LIN {X 0,Y 360.489,Z 777.93,A -85,B 0,C 180,E1 -13047.765,E2 -13047.765} C_VEL
LIN {X 0,Y 360.532,Z 778.599,A -85,B 0,C 180,E1 -13048.883,E2 -13048.883} C_VEL
LIN {X 0,Y 360.512,Z 778.865,A -85,B 0,C 180,E1 -13050,E2 -13050} C_VEL
LIN {X 0,Y 360.53,Z 778.734,A -85,B 0,C 180,E1 -13051.117,E2 -13051.117} C_VEL
LIN {X 0,Y 360.466,Z 778.154,A -85,B 0,C 180,E1 -13052.235,E2 -13052.235} C_VEL
LIN {X 0,Y 360.409,Z 775.773,A -85,B 0,C 180,E1 -13054.474,E2 -13054.474} C_VEL
LIN {X 0,Y 360.39,Z 773.205,A -85,B 0,C 180,E1 -13055.978,E2 -13055.978} C_VEL
LIN {X 0,Y 360.621,Z 768.887,A -85,B 0,C 180,E1 -13057.841,E2 -13057.841} C_VEL
LIN {X 0,Y 360.963,Z 763.784,A -85,B 0,C 180,E1 -13059.526,E2 -13059.526} C_VEL
LIN {X 0,Y 361.5,Z 757.4,A -85,B 0,C 180,E1 -13061.21,E2 -13061.21} C_VEL
LIN {X 0,Y 362.435,Z 749.451,A -85,B 0,C 180,E1 -13062.885,E2 -13062.885} C_VEL
LIN {X 0,Y 363.324,Z 741.358,A -85,B 0,C 180,E1 -13064.278,E2 -13064.278} C_VEL
LIN {X 0,Y 364.363,Z 731.514,A -85,B 0,C 180,E1 -13065.666,E2 -13065.666} C_VEL
LIN {X 0,Y 365.512,Z 720.605,A -85,B 0,C 180,E1 -13066.907,E2 -13066.907} C_VEL
LIN {X 0,Y 366.782,Z 708.229,A -85,B 0,C 180,E1 -13067.997,E2 -13067.997} C_VEL
LIN {X 0,Y 367.813,Z 696.177,A -85,B 0,C 180,E1 -13068.81,E2 -13068.81} C_VEL
LIN {X 0,Y 368.664,Z 683.917,A -85,B 0,C 180,E1 -13069.415,E2 -13069.415} C_VEL
LIN {X 0,Y 369.374,Z 670.122,A -85,B 0,C 180,E1 -13069.846,E2 -13069.846} C_VEL
LIN {X 0,Y 370.61,Z 601.907,A -85,B 0,C 180,E1 -13071.27,E2 -13071.27} C_VEL
LIN {X 0,Y 367.336,Z 578.506,A -85,B 0,C 180,E1 -13072.019,E2 -13072.019} C_VEL
LIN {X 0,Y 364.863,Z 564.206,A -85,B 0,C 180,E1 -13072.537,E2 -13072.537} C_VEL
LIN {X 0,Y 366.628,Z 547.673,A -85,B 0,C 180,E1 -13076.16,E2 -13076.16} C_VEL
LIN {X 0,Y 365.906,Z 542.347,A -85,B 0,C 180,E1 -13077.449,E2 -13077.449} C_VEL
LIN {X 0,Y 363.599,Z 531.727,A -85,B 0,C 180,E1 -13080.168,E2 -13080.168} C_VEL
LIN {X 0,Y 361.869,Z 524.409,A -85,B 0,C 180,E1 -13082.199,E2 -13082.199} C_VEL
LIN {X 0,Y 361.868,Z 524.412,A -85,B 0,C 180,E1 -13085.636,E2 -13085.636} C_VEL
LIN {X 0,Y 361.874,Z 524.408,A -85,B 0,C 180,E1 -13089.027,E2 -13089.027} C_VEL
LIN {X 0,Y 361.882,Z 524.409,A -85,B 0,C 180,E1 -13092.439,E2 -13092.439} C_VEL
LIN {X 0,Y 361.845,Z 524.41,A -85,B 0,C 180,E1 -13095.635,E2 -13095.635} C_VEL
LIN {X 0,Y 361.833,Z 524.412,A -85,B 0,C 180,E1 -13099.243,E2 -13099.243} C_VEL
LIN {X 0,Y 361.867,Z 524.407,A -85,B 0,C 180,E1 -13102.775,E2 -13102.775} C_VEL
LIN {X 0,Y 361.85,Z 524.406,A -85,B 0,C 180,E1 -13105.719,E2 -13105.719} C_VEL
LIN {X 0,Y 361.872,Z 524.405,A -85,B 0,C 180,E1 -13109.671,E2 -13109.671} C_VEL
LIN {X 0,Y 361.949,Z 524.398,A -85,B 0,C 180,E1 -13113.474,E2 -13113.474} C_VEL
LIN {X 0,Y 361.884,Z 524.408,A -85,B 0,C 180,E1 -13117.144,E2 -13117.144} C_VEL
LIN {X 0,Y 361.9,Z 524.405,A -85,B 0,C 180,E1 -13120.722,E2 -13120.722} C_VEL
LIN {X 0,Y 361.926,Z 524.398,A -85,B 0,C 180,E1 -13123.065,E2 -13123.065} C_VEL
LIN {X 0,Y 361.992,Z 524.389,A -85,B 0,C 180,E1 -13126.527,E2 -13126.527} C_VEL
LIN {X 0,Y 362.024,Z 524.383,A -85,B 0,C 180,E1 -13129.937,E2 -13129.937} C_VEL
LIN {X 0,Y 362.16,Z 524.367,A -85,B 0,C 180,E1 -13133.313,E2 -13133.313} C_VEL
LIN {X 0,Y 362.275,Z 524.355,A -85,B 0,C 180,E1 -13137.776,E2 -13137.776} C_VEL
LIN {X 0,Y 362.421,Z 524.336,A -85,B 0,C 180,E1 -13139.999,E2 -13139.999} C_VEL
LIN {X 0,Y 362.275,Z 524.357,A -85,B 0,C 180,E1 -13142.223,E2 -13142.223} C_VEL
LIN {X 0,Y 362.16,Z 524.37,A -85,B 0,C 180,E1 -13146.686,E2 -13146.686} C_VEL
LIN {X 0,Y 362.023,Z 524.389,A -85,B 0,C 180,E1 -13150.062,E2 -13150.062} C_VEL
LIN {X 0,Y 361.989,Z 524.393,A -85,B 0,C 180,E1 -13153.898,E2 -13153.898} C_VEL
LIN {X 0,Y 361.959,Z 524.398,A -85,B 0,C 180,E1 -13157.938,E2 -13157.938} C_VEL
LIN {X 0,Y 361.883,Z 524.409,A -85,B 0,C 180,E1 -13161.653,E2 -13161.653} C_VEL
LIN {X 0,Y 361.92,Z 524.407,A -85,B 0,C 180,E1 -13165.29,E2 -13165.29} C_VEL
LIN {X 0,Y 361.916,Z 524.444,A -85,B 0,C 180,E1 -13167.856,E2 -13167.856} C_VEL
LIN {X 0,Y 362.917,Z 529.129,A -85,B 0,C 180,E1 -13169.405,E2 -13169.405} C_VEL
LIN {X 0,Y 370.573,Z 547.908,A -85,B 0,C 180,E1 -13170.406,E2 -13170.406} C_VEL
LIN {X 0,Y 371.579,Z 551.185,A -85,B 0,C 180,E1 -13170.551,E2 -13170.551} C_VEL
LIN {X 0,Y 369.705,Z 635.83,A -85,B 0,C 180,E1 -13172.34,E2 -13172.34} C_VEL
LIN {X 0,Y 369.127,Z 649.318,A -85,B 0,C 180,E1 -13172.857,E2 -13172.857} C_VEL
LIN {X 0,Y 368.497,Z 661.898,A -85,B 0,C 180,E1 -13173.578,E2 -13173.578} C_VEL
LIN {X 0,Y 367.472,Z 674.408,A -85,B 0,C 180,E1 -13174.545,E2 -13174.545} C_VEL
LIN {X 0,Y 366.504,Z 685.226,A -85,B 0,C 180,E1 -13175.623,E2 -13175.623} C_VEL
LIN {X 0,Y 365.51,Z 694.463,A -85,B 0,C 180,E1 -13176.76,E2 -13176.76} C_VEL
LIN {X 0,Y 364.419,Z 703.419,A -85,B 0,C 180,E1 -13178.106,E2 -13178.106} C_VEL
LIN {X 0,Y 363.453,Z 711.718,A -85,B 0,C 180,E1 -13179.65,E2 -13179.65} C_VEL
LIN {X 0,Y 362.559,Z 718.622,A -85,B 0,C 180,E1 -13181.228,E2 -13181.228} C_VEL
LIN {X 0,Y 361.952,Z 724.194,A -85,B 0,C 180,E1 -13182.811,E2 -13182.811} C_VEL
LIN {X 0,Y 361.396,Z 728.754,A -85,B 0,C 180,E1 -13184.433,E2 -13184.433} C_VEL
LIN {X 0,Y 360.988,Z 732.319,A -85,B 0,C 180,E1 -13186.082,E2 -13186.082} C_VEL
LIN {X 0,Y 360.669,Z 734.956,A -85,B 0,C 180,E1 -13187.77,E2 -13187.77} C_VEL
LIN {X 0,Y 360.383,Z 736.968,A -85,B 0,C 180,E1 -13189.944,E2 -13189.944} C_VEL
LIN {X 0,Y 360.299,Z 737.425,A -85,B 0,C 180,E1 -13191.378,E2 -13191.378} C_VEL
LIN {X 0,Y 360.312,Z 737.13,A -85,B 0,C 180,E1 -13193.102,E2 -13193.102} C_VEL
LIN {X 0,Y 360.444,Z 735.727,A -85,B 0,C 180,E1 -13194.976,E2 -13194.976} C_VEL
LIN {X 0,Y 360.694,Z 733.029,A -85,B 0,C 180,E1 -13196.937,E2 -13196.937} C_VEL
LIN {X 0,Y 361.096,Z 728.94,A -85,B 0,C 180,E1 -13198.91,E2 -13198.91} C_VEL
LIN {X 0,Y 361.673,Z 722.976,A -85,B 0,C 180,E1 -13200.977,E2 -13200.977} C_VEL
LIN {X 0,Y 362.343,Z 716.425,A -85,B 0,C 180,E1 -13202.729,E2 -13202.729} C_VEL
LIN {X 0,Y 362.994,Z 709.72,A -85,B 0,C 180,E1 -13204.175,E2 -13204.175} C_VEL
LIN {X 0,Y 364.002,Z 700.212,A -85,B 0,C 180,E1 -13205.828,E2 -13205.828} C_VEL
LIN {X 0,Y 364.905,Z 690.474,A -85,B 0,C 180,E1 -13207.195,E2 -13207.195} C_VEL
LIN {X 0,Y 365.774,Z 680.843,A -85,B 0,C 180,E1 -13208.293,E2 -13208.293} C_VEL
LIN {X 0,Y 366.72,Z 668.626,A -85,B 0,C 180,E1 -13209.397,E2 -13209.397} C_VEL
LIN {X 0,Y 367.467,Z 656.612,A -85,B 0,C 180,E1 -13210.228,E2 -13210.228} C_VEL
LIN {X 0,Y 368.071,Z 643.724,A -85,B 0,C 180,E1 -13210.878,E2 -13210.878} C_VEL
LIN {X 0,Y 368.446,Z 630.868,A -85,B 0,C 180,E1 -13211.296,E2 -13211.296} C_VEL
LIN {X 0,Y 369.967,Z 550.083,A -85,B 0,C 180,E1 -13212.948,E2 -13212.948} C_VEL
LIN {X 0,Y 367.904,Z 542.538,A -85,B 0,C 180,E1 -13213.224,E2 -13213.224} C_VEL
LIN {X 0,Y 362.501,Z 527.124,A -85,B 0,C 180,E1 -13213.894,E2 -13213.894} C_VEL
LIN {X 0,Y 361.982,Z 524.398,A -85,B 0,C 180,E1 -13214.733,E2 -13214.733} C_VEL
LIN {X 0,Y 361.96,Z 524.394,A -85,B 0,C 180,E1 -13217.668,E2 -13217.668} C_VEL
LIN {X 0,Y 362.142,Z 524.371,A -85,B 0,C 180,E1 -13221.782,E2 -13221.782} C_VEL
LIN {X 0,Y 362.112,Z 524.377,A -85,B 0,C 180,E1 -13224.431,E2 -13224.431} C_VEL
LIN {X 0,Y 362.28,Z 524.354,A -85,B 0,C 180,E1 -13227.776,E2 -13227.776} C_VEL
LIN {X 0,Y 362.425,Z 524.336,A -85,B 0,C 180,E1 -13230,E2 -13230} C_VEL
LIN {X 0,Y 362.28,Z 524.355,A -85,B 0,C 180,E1 -13232.224,E2 -13232.224} C_VEL
LIN {X 0,Y 362.169,Z 524.372,A -85,B 0,C 180,E1 -13236.686,E2 -13236.686} C_VEL
LIN {X 0,Y 362.071,Z 524.387,A -85,B 0,C 180,E1 -13238.933,E2 -13238.933} C_VEL
LIN {X 0,Y 361.981,Z 524.391,A -85,B 0,C 180,E1 -13240.632,E2 -13240.632} C_VEL
LIN {X 0,Y 361.285,Z 524.482,A -85,B 0,C 180,E1 -13241.561,E2 -13241.561} C_VEL
LIN {X 0,Y 358.419,Z 524.841,A -85,B 0,C 180,E1 -13243.073,E2 -13243.073} C_VEL
LIN {X 0,Y 356.005,Z 525.141,A -85,B 0,C 180,E1 -13244.295,E2 -13244.295} C_VEL
LIN {X 0,Y 354.967,Z 525.269,A -85,B 0,C 180,E1 -13245.241,E2 -13245.241} C_VEL
LIN {X 0,Y 354.881,Z 525.276,A -85,B 0,C 180,E1 -13245.562,E2 -13245.562} C_VEL
LIN {X 0,Y 354.897,Z 525.275,A -85,B 0,C 180,E1 -13248.472,E2 -13248.472} C_VEL
LIN {X 0,Y 354.83,Z 525.282,A -85,B 0,C 180,E1 -13252.106,E2 -13252.106} C_VEL
LIN {X 0,Y 354.895,Z 525.274,A -85,B 0,C 180,E1 -13255.827,E2 -13255.827} C_VEL
LIN {X 0,Y 354.849,Z 525.28,A -85,B 0,C 180,E1 -13259.678,E2 -13259.678} C_VEL
LIN {X 0,Y 354.825,Z 525.284,A -85,B 0,C 180,E1 -13263.682,E2 -13263.682} C_VEL
LIN {X 0,Y 354.796,Z 525.288,A -85,B 0,C 180,E1 -13266.459,E2 -13266.459} C_VEL
LIN {X 0,Y 354.818,Z 525.286,A -85,B 0,C 180,E1 -13269.423,E2 -13269.423} C_VEL
LIN {X 0,Y 354.835,Z 525.286,A -85,B 0,C 180,E1 -13272.876,E2 -13272.876} C_VEL
LIN {X 0,Y 354.859,Z 525.279,A -85,B 0,C 180,E1 -13276.119,E2 -13276.119} C_VEL
LIN {X 0,Y 354.849,Z 525.285,A -85,B 0,C 180,E1 -13279.188,E2 -13279.188} C_VEL
LIN {X 0,Y 354.802,Z 525.286,A -85,B 0,C 180,E1 -13282.402,E2 -13282.402} C_VEL
LIN {X 0,Y 354.805,Z 525.29,A -85,B 0,C 180,E1 -13284.941,E2 -13284.941} C_VEL
LIN {X 0,Y 354.785,Z 525.288,A -85,B 0,C 180,E1 -13288.405,E2 -13288.405} C_VEL
LIN {X 0,Y 354.846,Z 525.282,A -85,B 0,C 180,E1 -13291.619,E2 -13291.619} C_VEL
LIN {X 0,Y 354.89,Z 525.275,A -85,B 0,C 180,E1 -13294.173,E2 -13294.173} C_VEL
LIN {X 0,Y 354.808,Z 525.285,A -85,B 0,C 180,E1 -13297.893,E2 -13297.893} C_VEL
LIN {X 0,Y 354.914,Z 525.272,A -85,B 0,C 180,E1 -13301.892,E2 -13301.892} C_VEL
LIN {X 0,Y 354.935,Z 525.269,A -85,B 0,C 180,E1 -13305.981,E2 -13305.981} C_VEL
LIN {X 0,Y 354.974,Z 525.265,A -85,B 0,C 180,E1 -13309.736,E2 -13309.736} C_VEL
LIN {X 0,Y 355.106,Z 525.248,A -85,B 0,C 180,E1 -13312.037,E2 -13312.037} C_VEL
LIN {X 0,Y 355.09,Z 525.25,A -85,B 0,C 180,E1 -13314.321,E2 -13314.321} C_VEL
LIN {X 0,Y 355.238,Z 525.233,A -85,B 0,C 180,E1 -13317.733,E2 -13317.733} C_VEL
LIN {X 0,Y 355.391,Z 525.213,A -85,B 0,C 180,E1 -13320.001,E2 -13320.001} C_VEL
LIN {X 0,Y 355.246,Z 525.23,A -85,B 0,C 180,E1 -13322.268,E2 -13322.268} C_VEL
LIN {X 0,Y 355.123,Z 525.248,A -85,B 0,C 180,E1 -13326.82,E2 -13326.82} C_VEL
LIN {X 0,Y 354.971,Z 525.265,A -85,B 0,C 180,E1 -13330.265,E2 -13330.265} C_VEL
LIN {X 0,Y 354.936,Z 525.269,A -85,B 0,C 180,E1 -13334.019,E2 -13334.019} C_VEL
LIN {X 0,Y 354.916,Z 525.272,A -85,B 0,C 180,E1 -13338.109,E2 -13338.109} C_VEL
LIN {X 0,Y 354.829,Z 525.282,A -85,B 0,C 180,E1 -13342.107,E2 -13342.107} C_VEL
LIN {X 0,Y 354.894,Z 525.276,A -85,B 0,C 180,E1 -13345.828,E2 -13345.828} C_VEL
LIN {X 0,Y 354.85,Z 525.282,A -85,B 0,C 180,E1 -13349.679,E2 -13349.679} C_VEL
LIN {X 0,Y 354.827,Z 525.285,A -85,B 0,C 180,E1 -13353.683,E2 -13353.683} C_VEL
LIN {X 0,Y 354.797,Z 525.286,A -85,B 0,C 180,E1 -13356.46,E2 -13356.46} C_VEL
LIN {X 0,Y 354.821,Z 525.289,A -85,B 0,C 180,E1 -13359.425,E2 -13359.425} C_VEL
LIN {X 0,Y 354.789,Z 525.289,A -85,B 0,C 180,E1 -13362.869,E2 -13362.869} C_VEL
LIN {X 0,Y 354.839,Z 525.281,A -85,B 0,C 180,E1 -13366.116,E2 -13366.116} C_VEL
LIN {X 0,Y 354.855,Z 525.284,A -85,B 0,C 180,E1 -13369.19,E2 -13369.19} C_VEL
LIN {X 0,Y 354.809,Z 525.285,A -85,B 0,C 180,E1 -13372.403,E2 -13372.403} C_VEL
LIN {X 0,Y 354.812,Z 525.286,A -85,B 0,C 180,E1 -13374.942,E2 -13374.942} C_VEL
LIN {X 0,Y 354.825,Z 525.36,A -85,B 0,C 180,E1 -13378.398,E2 -13378.398} C_VEL
LIN {X 0,Y 357.868,Z 539.227,A -85,B 0,C 180,E1 -13381.88,E2 -13381.88} C_VEL
LIN {X 0,Y 359.195,Z 546.187,A -85,B 0,C 180,E1 -13383.559,E2 -13383.559} C_VEL
LIN {X 0,Y 358.662,Z 553.068,A -85,B 0,C 180,E1 -13385.084,E2 -13385.084} C_VEL
LIN {X 0,Y 357.409,Z 565.665,A -85,B 0,C 180,E1 -13387.836,E2 -13387.836} C_VEL
LIN {X 0,Y 362.616,Z 603.252,A -85,B 0,C 180,E1 -13388.957,E2 -13388.957} C_VEL
LIN {X 0,Y 361.342,Z 674.648,A -85,B 0,C 180,E1 -13390.471,E2 -13390.471} C_VEL
LIN {X 0,Y 360.499,Z 688.367,A -85,B 0,C 180,E1 -13390.978,E2 -13390.978} C_VEL
LIN {X 0,Y 359.661,Z 700.264,A -85,B 0,C 180,E1 -13391.634,E2 -13391.634} C_VEL
LIN {X 0,Y 358.816,Z 711.594,A -85,B 0,C 180,E1 -13392.474,E2 -13392.474} C_VEL
LIN {X 0,Y 357.599,Z 723.289,A -85,B 0,C 180,E1 -13393.59,E2 -13393.59} C_VEL
LIN {X 0,Y 356.687,Z 733.434,A -85,B 0,C 180,E1 -13394.81,E2 -13394.81} C_VEL
LIN {X 0,Y 355.685,Z 743.354,A -85,B 0,C 180,E1 -13396.284,E2 -13396.284} C_VEL
LIN {X 0,Y 354.762,Z 752.511,A -85,B 0,C 180,E1 -13397.995,E2 -13397.995} C_VEL
LIN {X 0,Y 354.099,Z 759.888,A -85,B 0,C 180,E1 -13399.71,E2 -13399.71} C_VEL
LIN {X 0,Y 353.654,Z 765.787,A -85,B 0,C 180,E1 -13401.429,E2 -13401.429} C_VEL
LIN {X 0,Y 353.431,Z 770.417,A -85,B 0,C 180,E1 -13403.148,E2 -13403.148} C_VEL
LIN {X 0,Y 353.343,Z 772.847,A -85,B 0,C 180,E1 -13404.293,E2 -13404.293} C_VEL
LIN {X 0,Y 353.351,Z 774.835,A -85,B 0,C 180,E1 -13405.437,E2 -13405.437} C_VEL
LIN {X 0,Y 353.306,Z 776.391,A -85,B 0,C 180,E1 -13406.579,E2 -13406.579} C_VEL
LIN {X 0,Y 353.39,Z 777.496,A -85,B 0,C 180,E1 -13407.721,E2 -13407.721} C_VEL
LIN {X 0,Y 353.467,Z 778.176,A -85,B 0,C 180,E1 -13408.861,E2 -13408.861} C_VEL
LIN {X 0,Y 353.448,Z 778.451,A -85,B 0,C 180,E1 -13410,E2 -13410} C_VEL
LIN {X 0,Y 353.465,Z 778.33,A -85,B 0,C 180,E1 -13411.139,E2 -13411.139} C_VEL
LIN {X 0,Y 353.367,Z 777.762,A -85,B 0,C 180,E1 -13412.28,E2 -13412.28} C_VEL
LIN {X 0,Y 353.317,Z 775.399,A -85,B 0,C 180,E1 -13414.563,E2 -13414.563} C_VEL
LIN {X 0,Y 353.316,Z 773.108,A -85,B 0,C 180,E1 -13415.965,E2 -13415.965} C_VEL
LIN {X 0,Y 353.547,Z 768.557,A -85,B 0,C 180,E1 -13417.998,E2 -13417.998} C_VEL
LIN {X 0,Y 353.94,Z 763.482,A -85,B 0,C 180,E1 -13419.717,E2 -13419.717} C_VEL
LIN {X 0,Y 354.492,Z 757.119,A -85,B 0,C 180,E1 -13421.435,E2 -13421.435} C_VEL
LIN {X 0,Y 355.49,Z 749.214,A -85,B 0,C 180,E1 -13423.141,E2 -13423.141} C_VEL
LIN {X 0,Y 356.422,Z 741.154,A -85,B 0,C 180,E1 -13424.56,E2 -13424.56} C_VEL
LIN {X 0,Y 357.521,Z 731.349,A -85,B 0,C 180,E1 -13425.974,E2 -13425.974} C_VEL
LIN {X 0,Y 358.713,Z 720.496,A -85,B 0,C 180,E1 -13427.237,E2 -13427.237} C_VEL
LIN {X 0,Y 359.886,Z 709.991,A -85,B 0,C 180,E1 -13428.207,E2 -13428.207} C_VEL
LIN {X 0,Y 360.944,Z 698.556,A -85,B 0,C 180,E1 -13429.034,E2 -13429.034} C_VEL
LIN {X 0,Y 361.885,Z 685.825,A -85,B 0,C 180,E1 -13429.72,E2 -13429.72} C_VEL
LIN {X 0,Y 362.703,Z 672.672,A -85,B 0,C 180,E1 -13430.19,E2 -13430.19} C_VEL
LIN {X 0,Y 364.152,Z 603.214,A -85,B 0,C 180,E1 -13431.678,E2 -13431.678} C_VEL
LIN {X 0,Y 360.885,Z 579.589,A -85,B 0,C 180,E1 -13432.453,E2 -13432.453} C_VEL
LIN {X 0,Y 358.112,Z 563.696,A -85,B 0,C 180,E1 -13433.061,E2 -13433.061} C_VEL
LIN {X 0,Y 359.776,Z 548.549,A -85,B 0,C 180,E1 -13436.461,E2 -13436.461} C_VEL
LIN {X 0,Y 358.156,Z 539.568,A -85,B 0,C 180,E1 -13438.733,E2 -13438.733} C_VEL
LIN {X 0,Y 355.541,Z 528.262,A -85,B 0,C 180,E1 -13441.789,E2 -13441.789} C_VEL
LIN {X 0,Y 354.814,Z 525.287,A -85,B 0,C 180,E1 -13442.666,E2 -13442.666} C_VEL
LIN {X 0,Y 354.799,Z 525.294,A -85,B 0,C 180,E1 -13446.458,E2 -13446.458} C_VEL
LIN {X 0,Y 354.823,Z 525.287,A -85,B 0,C 180,E1 -13449.423,E2 -13449.423} C_VEL
LIN {X 0,Y 354.833,Z 525.284,A -85,B 0,C 180,E1 -13452.874,E2 -13452.874} C_VEL
LIN {X 0,Y 354.782,Z 525.29,A -85,B 0,C 180,E1 -13456.105,E2 -13456.105} C_VEL
LIN {X 0,Y 354.786,Z 525.291,A -85,B 0,C 180,E1 -13459.178,E2 -13459.178} C_VEL
LIN {X 0,Y 354.809,Z 525.288,A -85,B 0,C 180,E1 -13462.4,E2 -13462.4} C_VEL
LIN {X 0,Y 354.808,Z 525.288,A -85,B 0,C 180,E1 -13464.94,E2 -13464.94} C_VEL
LIN {X 0,Y 354.789,Z 525.291,A -85,B 0,C 180,E1 -13468.404,E2 -13468.404} C_VEL
LIN {X 0,Y 354.849,Z 525.279,A -85,B 0,C 180,E1 -13471.618,E2 -13471.618} C_VEL
LIN {X 0,Y 354.894,Z 525.277,A -85,B 0,C 180,E1 -13474.172,E2 -13474.172} C_VEL
LIN {X 0,Y 354.829,Z 525.284,A -85,B 0,C 180,E1 -13477.893,E2 -13477.893} C_VEL
LIN {X 0,Y 354.916,Z 525.272,A -85,B 0,C 180,E1 -13481.891,E2 -13481.891} C_VEL
LIN {X 0,Y 354.936,Z 525.268,A -85,B 0,C 180,E1 -13485.981,E2 -13485.981} C_VEL
LIN {X 0,Y 354.971,Z 525.262,A -85,B 0,C 180,E1 -13489.735,E2 -13489.735} C_VEL
LIN {X 0,Y 355.124,Z 525.245,A -85,B 0,C 180,E1 -13493.18,E2 -13493.18} C_VEL
LIN {X 0,Y 355.238,Z 525.232,A -85,B 0,C 180,E1 -13497.732,E2 -13497.732} C_VEL
LIN {X 0,Y 355.391,Z 525.212,A -85,B 0,C 180,E1 -13499.999,E2 -13499.999} C_VEL
LIN {X 0,Y 355.239,Z 525.234,A -85,B 0,C 180,E1 -13502.267,E2 -13502.267} C_VEL
LIN {X 0,Y 355.122,Z 525.247,A -85,B 0,C 180,E1 -13506.819,E2 -13506.819} C_VEL
LIN {X 0,Y 354.97,Z 525.268,A -85,B 0,C 180,E1 -13510.264,E2 -13510.264} C_VEL
LIN {X 0,Y 354.934,Z 525.272,A -85,B 0,C 180,E1 -13514.018,E2 -13514.018} C_VEL
LIN {X 0,Y 354.914,Z 525.275,A -85,B 0,C 180,E1 -13518.108,E2 -13518.108} C_VEL
LIN {X 0,Y 354.826,Z 525.288,A -85,B 0,C 180,E1 -13522.106,E2 -13522.106} C_VEL
LIN {X 0,Y 354.891,Z 525.286,A -85,B 0,C 180,E1 -13525.827,E2 -13525.827} C_VEL
LIN {X 0,Y 354.881,Z 525.353,A -85,B 0,C 180,E1 -13527.415,E2 -13527.415} C_VEL
LIN {X 0,Y 355.808,Z 529.629,A -85,B 0,C 180,E1 -13528.861,E2 -13528.861} C_VEL
LIN {X 0,Y 364.058,Z 549.422,A -85,B 0,C 180,E1 -13529.972,E2 -13529.972} C_VEL
LIN {X 0,Y 365.108,Z 552.979,A -85,B 0,C 180,E1 -13530.13,E2 -13530.13} C_VEL
LIN {X 0,Y 363.179,Z 635.861,A -85,B 0,C 180,E1 -13531.912,E2 -13531.912} C_VEL
LIN {X 0,Y 362.54,Z 649.631,A -85,B 0,C 180,E1 -13532.445,E2 -13532.445} C_VEL
LIN {X 0,Y 361.85,Z 662.534,A -85,B 0,C 180,E1 -13533.2,E2 -13533.2} C_VEL
LIN {X 0,Y 360.885,Z 674.159,A -85,B 0,C 180,E1 -13534.112,E2 -13534.112} C_VEL
LIN {X 0,Y 359.816,Z 685.371,A -85,B 0,C 180,E1 -13535.24,E2 -13535.24} C_VEL
LIN {X 0,Y 358.654,Z 695.705,A -85,B 0,C 180,E1 -13536.544,E2 -13536.544} C_VEL
LIN {X 0,Y 357.402,Z 705.748,A -85,B 0,C 180,E1 -13538.136,E2 -13538.136} C_VEL
LIN {X 0,Y 356.366,Z 713.816,A -85,B 0,C 180,E1 -13539.726,E2 -13539.726} C_VEL
LIN {X 0,Y 355.488,Z 720.292,A -85,B 0,C 180,E1 -13541.302,E2 -13541.302} C_VEL
LIN {X 0,Y 354.864,Z 725.527,A -85,B 0,C 180,E1 -13542.882,E2 -13542.882} C_VEL
LIN {X 0,Y 354.328,Z 729.648,A -85,B 0,C 180,E1 -13544.436,E2 -13544.436} C_VEL
LIN {X 0,Y 353.934,Z 732.832,A -85,B 0,C 180,E1 -13545.975,E2 -13545.975} C_VEL
LIN {X 0,Y 353.632,Z 735.186,A -85,B 0,C 180,E1 -13547.492,E2 -13547.492} C_VEL
LIN {X 0,Y 353.387,Z 736.867,A -85,B 0,C 180,E1 -13549.088,E2 -13549.088} C_VEL
LIN {X 0,Y 353.225,Z 737.791,A -85,B 0,C 180,E1 -13550.892,E2 -13550.892} C_VEL
LIN {X 0,Y 353.222,Z 737.698,A -85,B 0,C 180,E1 -13552.737,E2 -13552.737} C_VEL
LIN {X 0,Y 353.33,Z 736.363,A -85,B 0,C 180,E1 -13554.773,E2 -13554.773} C_VEL
LIN {X 0,Y 353.527,Z 734.055,A -85,B 0,C 180,E1 -13556.609,E2 -13556.609} C_VEL
LIN {X 0,Y 353.967,Z 730.222,A -85,B 0,C 180,E1 -13558.622,E2 -13558.622} C_VEL
LIN {X 0,Y 354.345,Z 725.964,A -85,B 0,C 180,E1 -13560.275,E2 -13560.275} C_VEL
LIN {X 0,Y 355.07,Z 719.266,A -85,B 0,C 180,E1 -13562.282,E2 -13562.282} C_VEL
LIN {X 0,Y 355.832,Z 712.229,A -85,B 0,C 180,E1 -13563.931,E2 -13563.931} C_VEL
LIN {X 0,Y 356.746,Z 703.616,A -85,B 0,C 180,E1 -13565.563,E2 -13565.563} C_VEL
LIN {X 0,Y 357.725,Z 694.207,A -85,B 0,C 180,E1 -13567.006,E2 -13567.006} C_VEL
LIN {X 0,Y 358.662,Z 683.745,A -85,B 0,C 180,E1 -13568.294,E2 -13568.294} C_VEL
LIN {X 0,Y 359.646,Z 672.39,A -85,B 0,C 180,E1 -13569.406,E2 -13569.406} C_VEL
LIN {X 0,Y 360.479,Z 659.888,A -85,B 0,C 180,E1 -13570.356,E2 -13570.356} C_VEL
LIN {X 0,Y 361.132,Z 646.613,A -85,B 0,C 180,E1 -13571.087,E2 -13571.087} C_VEL
LIN {X 0,Y 361.607,Z 633.983,A -85,B 0,C 180,E1 -13571.553,E2 -13571.553} C_VEL
LIN {X 0,Y 363.192,Z 550.766,A -85,B 0,C 180,E1 -13573.308,E2 -13573.308} C_VEL
LIN {X 0,Y 359.766,Z 539.781,A -85,B 0,C 180,E1 -13573.747,E2 -13573.747} C_VEL
LIN {X 0,Y 355.361,Z 527.561,A -85,B 0,C 180,E1 -13574.295,E2 -13574.295} C_VEL
LIN {X 0,Y 354.915,Z 525.276,A -85,B 0,C 180,E1 -13575.01,E2 -13575.01} C_VEL
LIN {X 0,Y 354.932,Z 525.273,A -85,B 0,C 180,E1 -13578.58,E2 -13578.58} C_VEL
LIN {X 0,Y 355.081,Z 525.251,A -85,B 0,C 180,E1 -13582.036,E2 -13582.036} C_VEL
LIN {X 0,Y 355.086,Z 525.251,A -85,B 0,C 180,E1 -13584.321,E2 -13584.321} C_VEL
LIN {X 0,Y 355.243,Z 525.231,A -85,B 0,C 180,E1 -13587.732,E2 -13587.732} C_VEL
LIN {X 0,Y 355.395,Z 525.212,A -85,B 0,C 180,E1 -13590,E2 -13590} C_VEL
LIN {X 0,Y 355.243,Z 525.231,A -85,B 0,C 180,E1 -13592.268,E2 -13592.268} C_VEL
LIN {X 0,Y 355.135,Z 525.249,A -85,B 0,C 180,E1 -13596.819,E2 -13596.819} C_VEL
LIN {X 0,Y 355.012,Z 525.264,A -85,B 0,C 180,E1 -13599.112,E2 -13599.112} C_VEL
LIN {X 0,Y 354.918,Z 525.274,A -85,B 0,C 180,E1 -13602.581,E2 -13602.581} C_VEL
LIN {X 0,Y 354.881,Z 525.276,A -85,B 0,C 180,E1 -13605.562,E2 -13605.562} C_VEL
LIN {X 0,Y 354.204,Z 525.364,A -85,B 0,C 180,E1 -13606.51,E2 -13606.51} C_VEL
LIN {X 0,Y 351.337,Z 525.717,A -85,B 0,C 180,E1 -13608.052,E2 -13608.052} C_VEL
LIN {X 0,Y 348.913,Z 526.022,A -85,B 0,C 180,E1 -13609.299,E2 -13609.299} C_VEL
LIN {X 0,Y 347.875,Z 526.149,A -85,B 0,C 180,E1 -13610.265,E2 -13610.265} C_VEL
LIN {X 0,Y 347.792,Z 526.158,A -85,B 0,C 180,E1 -13610.592,E2 -13610.592} C_VEL
LIN {X 0,Y 347.812,Z 526.159,A -85,B 0,C 180,E1 -13614.595,E2 -13614.595} C_VEL
LIN {X 0,Y 347.808,Z 526.158,A -85,B 0,C 180,E1 -13617.693,E2 -13617.693} C_VEL
LIN {X 0,Y 347.766,Z 526.163,A -85,B 0,C 180,E1 -13620.345,E2 -13620.345} C_VEL
LIN {X 0,Y 347.743,Z 526.165,A -85,B 0,C 180,E1 -13624.044,E2 -13624.044} C_VEL
LIN {X 0,Y 347.761,Z 526.166,A -85,B 0,C 180,E1 -13627.32,E2 -13627.32} C_VEL
LIN {X 0,Y 347.787,Z 526.16,A -85,B 0,C 180,E1 -13630.288,E2 -13630.288} C_VEL
LIN {X 0,Y 347.812,Z 526.159,A -85,B 0,C 180,E1 -13633.393,E2 -13633.393} C_VEL
LIN {X 0,Y 347.81,Z 526.159,A -85,B 0,C 180,E1 -13636.67,E2 -13636.67} C_VEL
LIN {X 0,Y 347.778,Z 526.161,A -85,B 0,C 180,E1 -13640.165,E2 -13640.165} C_VEL
LIN {X 0,Y 347.781,Z 526.16,A -85,B 0,C 180,E1 -13644.125,E2 -13644.125} C_VEL
LIN {X 0,Y 347.731,Z 526.167,A -85,B 0,C 180,E1 -13648.086,E2 -13648.086} C_VEL
LIN {X 0,Y 347.799,Z 526.163,A -85,B 0,C 180,E1 -13650.99,E2 -13650.99} C_VEL
LIN {X 0,Y 347.823,Z 526.157,A -85,B 0,C 180,E1 -13653.608,E2 -13653.608} C_VEL
LIN {X 0,Y 347.777,Z 526.161,A -85,B 0,C 180,E1 -13656.162,E2 -13656.162} C_VEL
LIN {X 0,Y 347.798,Z 526.159,A -85,B 0,C 180,E1 -13659.909,E2 -13659.909} C_VEL
LIN {X 0,Y 347.858,Z 526.151,A -85,B 0,C 180,E1 -13662.359,E2 -13662.359} C_VEL
LIN {X 0,Y 347.889,Z 526.147,A -85,B 0,C 180,E1 -13665.971,E2 -13665.971} C_VEL
LIN {X 0,Y 347.925,Z 526.145,A -85,B 0,C 180,E1 -13669.526,E2 -13669.526} C_VEL
LIN {X 0,Y 348.066,Z 526.125,A -85,B 0,C 180,E1 -13671.875,E2 -13671.875} C_VEL
LIN {X 0,Y 348.065,Z 526.125,A -85,B 0,C 180,E1 -13674.206,E2 -13674.206} C_VEL
LIN {X 0,Y 348.201,Z 526.11,A -85,B 0,C 180,E1 -13677.687,E2 -13677.687} C_VEL
LIN {X 0,Y 348.361,Z 526.088,A -85,B 0,C 180,E1 -13680.001,E2 -13680.001} C_VEL
LIN {X 0,Y 348.209,Z 526.107,A -85,B 0,C 180,E1 -13682.314,E2 -13682.314} C_VEL
LIN {X 0,Y 348.088,Z 526.126,A -85,B 0,C 180,E1 -13686.959,E2 -13686.959} C_VEL
LIN {X 0,Y 347.922,Z 526.143,A -85,B 0,C 180,E1 -13690.475,E2 -13690.475} C_VEL
LIN {X 0,Y 347.892,Z 526.146,A -85,B 0,C 180,E1 -13694.151,E2 -13694.151} C_VEL
LIN {X 0,Y 347.884,Z 526.147,A -85,B 0,C 180,E1 -13698.291,E2 -13698.291} C_VEL
LIN {X 0,Y 347.783,Z 526.163,A -85,B 0,C 180,E1 -13701.636,E2 -13701.636} C_VEL
LIN {X 0,Y 347.807,Z 526.161,A -85,B 0,C 180,E1 -13705.109,E2 -13705.109} C_VEL
LIN {X 0,Y 347.807,Z 526.159,A -85,B 0,C 180,E1 -13707.695,E2 -13707.695} C_VEL
LIN {X 0,Y 347.766,Z 526.162,A -85,B 0,C 180,E1 -13710.347,E2 -13710.347} C_VEL
LIN {X 0,Y 347.744,Z 526.165,A -85,B 0,C 180,E1 -13714.045,E2 -13714.045} C_VEL
LIN {X 0,Y 347.762,Z 526.169,A -85,B 0,C 180,E1 -13717.321,E2 -13717.321} C_VEL
LIN {X 0,Y 347.73,Z 526.167,A -85,B 0,C 180,E1 -13720.298,E2 -13720.298} C_VEL
LIN {X 0,Y 347.727,Z 526.173,A -85,B 0,C 180,E1 -13723.408,E2 -13723.408} C_VEL
LIN {X 0,Y 347.781,Z 526.161,A -85,B 0,C 180,E1 -13726.677,E2 -13726.677} C_VEL
LIN {X 0,Y 347.785,Z 526.16,A -85,B 0,C 180,E1 -13730.166,E2 -13730.166} C_VEL
LIN {X 0,Y 347.789,Z 526.16,A -85,B 0,C 180,E1 -13734.126,E2 -13734.126} C_VEL
LIN {X 0,Y 347.784,Z 526.305,A -85,B 0,C 180,E1 -13738.075,E2 -13738.075} C_VEL
LIN {X 0,Y 350.807,Z 540.039,A -85,B 0,C 180,E1 -13741.604,E2 -13741.604} C_VEL
LIN {X 0,Y 352.273,Z 548.524,A -85,B 0,C 180,E1 -13743.68,E2 -13743.68} C_VEL
LIN {X 0,Y 350.822,Z 562.85,A -85,B 0,C 180,E1 -13746.888,E2 -13746.888} C_VEL
LIN {X 0,Y 350.562,Z 565.347,A -85,B 0,C 180,E1 -13747.432,E2 -13747.432} C_VEL
LIN {X 0,Y 355.879,Z 604.297,A -85,B 0,C 180,E1 -13748.621,E2 -13748.621} C_VEL
LIN {X 0,Y 354.529,Z 674.942,A -85,B 0,C 180,E1 -13750.156,E2 -13750.156} C_VEL
LIN {X 0,Y 353.676,Z 688.432,A -85,B 0,C 180,E1 -13750.672,E2 -13750.672} C_VEL
LIN {X 0,Y 352.828,Z 700.21,A -85,B 0,C 180,E1 -13751.341,E2 -13751.341} C_VEL
LIN {X 0,Y 351.864,Z 712.234,A -85,B 0,C 180,E1 -13752.266,E2 -13752.266} C_VEL
LIN {X 0,Y 350.61,Z 723.739,A -85,B 0,C 180,E1 -13753.403,E2 -13753.403} C_VEL
LIN {X 0,Y 349.693,Z 733.488,A -85,B 0,C 180,E1 -13754.613,E2 -13754.613} C_VEL
LIN {X 0,Y 348.765,Z 742.666,A -85,B 0,C 180,E1 -13756.007,E2 -13756.007} C_VEL
LIN {X 0,Y 347.756,Z 751.879,A -85,B 0,C 180,E1 -13757.749,E2 -13757.749} C_VEL
LIN {X 0,Y 347.042,Z 759.3,A -85,B 0,C 180,E1 -13759.499,E2 -13759.499} C_VEL
LIN {X 0,Y 346.61,Z 765.244,A -85,B 0,C 180,E1 -13761.253,E2 -13761.253} C_VEL
LIN {X 0,Y 346.374,Z 769.91,A -85,B 0,C 180,E1 -13763.008,E2 -13763.008} C_VEL
LIN {X 0,Y 346.233,Z 773.438,A -85,B 0,C 180,E1 -13764.759,E2 -13764.759} C_VEL
LIN {X 0,Y 346.226,Z 775.931,A -85,B 0,C 180,E1 -13766.509,E2 -13766.509} C_VEL
LIN {X 0,Y 346.293,Z 777.058,A -85,B 0,C 180,E1 -13767.674,E2 -13767.674} C_VEL
LIN {X 0,Y 346.385,Z 777.749,A -85,B 0,C 180,E1 -13768.837,E2 -13768.837} C_VEL
LIN {X 0,Y 346.385,Z 778.036,A -85,B 0,C 180,E1 -13770,E2 -13770} C_VEL
LIN {X 0,Y 346.382,Z 777.924,A -85,B 0,C 180,E1 -13771.163,E2 -13771.163} C_VEL
LIN {X 0,Y 346.268,Z 777.377,A -85,B 0,C 180,E1 -13772.326,E2 -13772.326} C_VEL
LIN {X 0,Y 346.229,Z 775.033,A -85,B 0,C 180,E1 -13774.657,E2 -13774.657} C_VEL
LIN {X 0,Y 346.283,Z 772.153,A -85,B 0,C 180,E1 -13776.408,E2 -13776.408} C_VEL
LIN {X 0,Y 346.496,Z 768.232,A -85,B 0,C 180,E1 -13778.162,E2 -13778.162} C_VEL
LIN {X 0,Y 346.902,Z 763.177,A -85,B 0,C 180,E1 -13779.916,E2 -13779.916} C_VEL
LIN {X 0,Y 347.502,Z 756.839,A -85,B 0,C 180,E1 -13781.668,E2 -13781.668} C_VEL
LIN {X 0,Y 348.546,Z 748.977,A -85,B 0,C 180,E1 -13783.408,E2 -13783.408} C_VEL
LIN {X 0,Y 349.696,Z 739.148,A -85,B 0,C 180,E1 -13785.145,E2 -13785.145} C_VEL
LIN {X 0,Y 350.924,Z 729.051,A -85,B 0,C 180,E1 -13786.582,E2 -13786.582} C_VEL
LIN {X 0,Y 352.27,Z 717.674,A -85,B 0,C 180,E1 -13787.862,E2 -13787.862} C_VEL
LIN {X 0,Y 353.452,Z 706.582,A -85,B 0,C 180,E1 -13788.851,E2 -13788.851} C_VEL
LIN {X 0,Y 354.595,Z 694.349,A -85,B 0,C 180,E1 -13789.69,E2 -13789.69} C_VEL
LIN {X 0,Y 355.588,Z 681.588,A -85,B 0,C 180,E1 -13790.31,E2 -13790.31} C_VEL
LIN {X 0,Y 356.272,Z 668.433,A -85,B 0,C 180,E1 -13790.722,E2 -13790.722} C_VEL
LIN {X 0,Y 357.575,Z 603.339,A -85,B 0,C 180,E1 -13792.14,E2 -13792.14} C_VEL
LIN {X 0,Y 354.137,Z 578.578,A -85,B 0,C 180,E1 -13792.98,E2 -13792.98} C_VEL
LIN {X 0,Y 351.35,Z 563.309,A -85,B 0,C 180,E1 -13793.581,E2 -13793.581} C_VEL
LIN {X 0,Y 352.879,Z 549.82,A -85,B 0,C 180,E1 -13796.682,E2 -13796.682} C_VEL
LIN {X 0,Y 350.929,Z 539.488,A -85,B 0,C 180,E1 -13799.383,E2 -13799.383} C_VEL
LIN {X 0,Y 348.062,Z 527.452,A -85,B 0,C 180,E1 -13802.766,E2 -13802.766} C_VEL
LIN {X 0,Y 347.783,Z 526.166,A -85,B 0,C 180,E1 -13803.147,E2 -13803.147} C_VEL
LIN {X 0,Y 347.771,Z 526.168,A -85,B 0,C 180,E1 -13806.064,E2 -13806.064} C_VEL
LIN {X 0,Y 347.785,Z 526.164,A -85,B 0,C 180,E1 -13809.834,E2 -13809.834} C_VEL
LIN {X 0,Y 347.784,Z 526.163,A -85,B 0,C 180,E1 -13813.397,E2 -13813.397} C_VEL
LIN {X 0,Y 347.728,Z 526.172,A -85,B 0,C 180,E1 -13816.684,E2 -13816.684} C_VEL
LIN {X 0,Y 347.744,Z 526.165,A -85,B 0,C 180,E1 -13820.172,E2 -13820.172} C_VEL
LIN {X 0,Y 347.762,Z 526.164,A -85,B 0,C 180,E1 -13822.679,E2 -13822.679} C_VEL
LIN {X 0,Y 347.744,Z 526.163,A -85,B 0,C 180,E1 -13825.955,E2 -13825.955} C_VEL
LIN {X 0,Y 347.76,Z 526.163,A -85,B 0,C 180,E1 -13829.653,E2 -13829.653} C_VEL
LIN {X 0,Y 347.848,Z 526.152,A -85,B 0,C 180,E1 -13832.743,E2 -13832.743} C_VEL
LIN {X 0,Y 347.783,Z 526.156,A -85,B 0,C 180,E1 -13836.161,E2 -13836.161} C_VEL
LIN {X 0,Y 347.806,Z 526.156,A -85,B 0,C 180,E1 -13839.908,E2 -13839.908} C_VEL
LIN {X 0,Y 347.86,Z 526.151,A -85,B 0,C 180,E1 -13842.358,E2 -13842.358} C_VEL
LIN {X 0,Y 347.891,Z 526.146,A -85,B 0,C 180,E1 -13845.97,E2 -13845.97} C_VEL
LIN {X 0,Y 347.922,Z 526.141,A -85,B 0,C 180,E1 -13849.525,E2 -13849.525} C_VEL
LIN {X 0,Y 348.089,Z 526.122,A -85,B 0,C 180,E1 -13853.041,E2 -13853.041} C_VEL
LIN {X 0,Y 348.201,Z 526.109,A -85,B 0,C 180,E1 -13857.686,E2 -13857.686} C_VEL
LIN {X 0,Y 348.361,Z 526.087,A -85,B 0,C 180,E1 -13859.999,E2 -13859.999} C_VEL
LIN {X 0,Y 348.201,Z 526.111,A -85,B 0,C 180,E1 -13862.313,E2 -13862.313} C_VEL
LIN {X 0,Y 348.087,Z 526.124,A -85,B 0,C 180,E1 -13866.957,E2 -13866.957} C_VEL
LIN {X 0,Y 347.92,Z 526.147,A -85,B 0,C 180,E1 -13870.474,E2 -13870.474} C_VEL
LIN {X 0,Y 347.89,Z 526.149,A -85,B 0,C 180,E1 -13874.15,E2 -13874.15} C_VEL
LIN {X 0,Y 347.882,Z 526.151,A -85,B 0,C 180,E1 -13878.29,E2 -13878.29} C_VEL
LIN {X 0,Y 347.78,Z 526.166,A -85,B 0,C 180,E1 -13881.635,E2 -13881.635} C_VEL
LIN {X 0,Y 347.804,Z 526.164,A -85,B 0,C 180,E1 -13885.108,E2 -13885.108} C_VEL
LIN {X 0,Y 347.837,Z 526.259,A -85,B 0,C 180,E1 -13886.94,E2 -13886.94} C_VEL
LIN {X 0,Y 348.771,Z 530.36,A -85,B 0,C 180,E1 -13888.305,E2 -13888.305} C_VEL
LIN {X 0,Y 357.168,Z 550.02,A -85,B 0,C 180,E1 -13889.467,E2 -13889.467} C_VEL
LIN {X 0,Y 358.543,Z 553.771,A -85,B 0,C 180,E1 -13889.663,E2 -13889.663} C_VEL
LIN {X 0,Y 356.634,Z 636.32,A -85,B 0,C 180,E1 -13891.481,E2 -13891.481} C_VEL
LIN {X 0,Y 355.964,Z 650.15,A -85,B 0,C 180,E1 -13892.026,E2 -13892.026} C_VEL
LIN {X 0,Y 355.265,Z 662.916,A -85,B 0,C 180,E1 -13892.788,E2 -13892.788} C_VEL
LIN {X 0,Y 354.217,Z 674.908,A -85,B 0,C 180,E1 -13893.748,E2 -13893.748} C_VEL
LIN {X 0,Y 353.113,Z 685.911,A -85,B 0,C 180,E1 -13894.878,E2 -13894.878} C_VEL
LIN {X 0,Y 351.976,Z 695.412,A -85,B 0,C 180,E1 -13896.088,E2 -13896.088} C_VEL
LIN {X 0,Y 350.642,Z 705.411,A -85,B 0,C 180,E1 -13897.677,E2 -13897.677} C_VEL
LIN {X 0,Y 349.577,Z 713.538,A -85,B 0,C 180,E1 -13899.286,E2 -13899.286} C_VEL
LIN {X 0,Y 348.623,Z 720.166,A -85,B 0,C 180,E1 -13900.9,E2 -13900.9} C_VEL
LIN {X 0,Y 347.784,Z 726.675,A -85,B 0,C 180,E1 -13902.918,E2 -13902.918} C_VEL
LIN {X 0,Y 347.104,Z 731.967,A -85,B 0,C 180,E1 -13905.125,E2 -13905.125} C_VEL
LIN {X 0,Y 346.67,Z 734.948,A -85,B 0,C 180,E1 -13906.871,E2 -13906.871} C_VEL
LIN {X 0,Y 346.358,Z 736.993,A -85,B 0,C 180,E1 -13908.656,E2 -13908.656} C_VEL
LIN {X 0,Y 346.132,Z 738.225,A -85,B 0,C 180,E1 -13910.993,E2 -13910.993} C_VEL
LIN {X 0,Y 346.123,Z 738.167,A -85,B 0,C 180,E1 -13912.473,E2 -13912.473} C_VEL
LIN {X 0,Y 346.199,Z 737.206,A -85,B 0,C 180,E1 -13914.292,E2 -13914.292} C_VEL
LIN {X 0,Y 346.39,Z 735.024,A -85,B 0,C 180,E1 -13916.289,E2 -13916.289} C_VEL
LIN {X 0,Y 346.814,Z 731.451,A -85,B 0,C 180,E1 -13918.331,E2 -13918.331} C_VEL
LIN {X 0,Y 347.337,Z 726.176,A -85,B 0,C 180,E1 -13920.464,E2 -13920.464} C_VEL
LIN {X 0,Y 348.001,Z 720.119,A -85,B 0,C 180,E1 -13922.323,E2 -13922.323} C_VEL
LIN {X 0,Y 348.791,Z 713.176,A -85,B 0,C 180,E1 -13924.008,E2 -13924.008} C_VEL
LIN {X 0,Y 349.712,Z 704.675,A -85,B 0,C 180,E1 -13925.671,E2 -13925.671} C_VEL
LIN {X 0,Y 350.747,Z 695.169,A -85,B 0,C 180,E1 -13927.176,E2 -13927.176} C_VEL
LIN {X 0,Y 351.684,Z 685.162,A -85,B 0,C 180,E1 -13928.457,E2 -13928.457} C_VEL
LIN {X 0,Y 352.744,Z 673.711,A -85,B 0,C 180,E1 -13929.619,E2 -13929.619} C_VEL
LIN {X 0,Y 353.573,Z 661.992,A -85,B 0,C 180,E1 -13930.553,E2 -13930.553} C_VEL
LIN {X 0,Y 354.292,Z 649.216,A -85,B 0,C 180,E1 -13931.308,E2 -13931.308} C_VEL
LIN {X 0,Y 354.821,Z 635.674,A -85,B 0,C 180,E1 -13931.848,E2 -13931.848} C_VEL
LIN {X 0,Y 355.84,Z 588.088,A -85,B 0,C 180,E1 -13932.888,E2 -13932.888} C_VEL
LIN {X 0,Y 356.527,Z 551.911,A -85,B 0,C 180,E1 -13933.661,E2 -13933.661} C_VEL
LIN {X 0,Y 350.987,Z 535.554,A -85,B 0,C 180,E1 -13934.363,E2 -13934.363} C_VEL
LIN {X 0,Y 348.23,Z 527.955,A -85,B 0,C 180,E1 -13934.722,E2 -13934.722} C_VEL
LIN {X 0,Y 347.909,Z 526.146,A -85,B 0,C 180,E1 -13935.3,E2 -13935.3} C_VEL
LIN {X 0,Y 347.882,Z 526.149,A -85,B 0,C 180,E1 -13938.345,E2 -13938.345} C_VEL
LIN {X 0,Y 348.043,Z 526.128,A -85,B 0,C 180,E1 -13941.874,E2 -13941.874} C_VEL
LIN {X 0,Y 348.06,Z 526.126,A -85,B 0,C 180,E1 -13944.206,E2 -13944.206} C_VEL
LIN {X 0,Y 348.206,Z 526.108,A -85,B 0,C 180,E1 -13947.687,E2 -13947.687} C_VEL
LIN {X 0,Y 348.344,Z 526.09,A -85,B 0,C 180,E1 -13950,E2 -13950} C_VEL
LIN {X 0,Y 348.205,Z 526.108,A -85,B 0,C 180,E1 -13952.313,E2 -13952.313} C_VEL
LIN {X 0,Y 348.104,Z 526.126,A -85,B 0,C 180,E1 -13956.958,E2 -13956.958} C_VEL
LIN {X 0,Y 347.964,Z 526.14,A -85,B 0,C 180,E1 -13959.298,E2 -13959.298} C_VEL
LIN {X 0,Y 347.886,Z 526.152,A -85,B 0,C 180,E1 -13962.839,E2 -13962.839} C_VEL
LIN {X 0,Y 347.835,Z 526.155,A -85,B 0,C 180,E1 -13966.431,E2 -13966.431} C_VEL
LIN {X 0,Y 347.847,Z 526.157,A -85,B 0,C 180,E1 -13968.86,E2 -13968.86} C_VEL
LIN {X 0,Y 347.792,Z 526.158,A -85,B 0,C 180,E1 -13970.592,E2 -13970.592} C_VEL
LIN {X 0,Y 347.136,Z 526.243,A -85,B 0,C 180,E1 -13971.558,E2 -13971.558} C_VEL
LIN {X 0,Y 344.31,Z 526.598,A -85,B 0,C 180,E1 -13973.129,E2 -13973.129} C_VEL
LIN {X 0,Y 341.904,Z 526.897,A -85,B 0,C 180,E1 -13974.401,E2 -13974.401} C_VEL
LIN {X 0,Y 340.858,Z 527.026,A -85,B 0,C 180,E1 -13975.385,E2 -13975.385} C_VEL
LIN {X 0,Y 340.766,Z 527.035,A -85,B 0,C 180,E1 -13975.718,E2 -13975.718} C_VEL
LIN {X 0,Y 340.738,Z 527.038,A -85,B 0,C 180,E1 -13978.319,E2 -13978.319} C_VEL
LIN {X 0,Y 340.711,Z 527.047,A -85,B 0,C 180,E1 -13981.042,E2 -13981.042} C_VEL
LIN {X 0,Y 340.713,Z 527.044,A -85,B 0,C 180,E1 -13985.278,E2 -13985.278} C_VEL
LIN {X 0,Y 340.714,Z 527.041,A -85,B 0,C 180,E1 -13988.388,E2 -13988.388} C_VEL
LIN {X 0,Y 340.72,Z 527.044,A -85,B 0,C 180,E1 -13991.303,E2 -13991.303} C_VEL
LIN {X 0,Y 340.774,Z 527.034,A -85,B 0,C 180,E1 -13994.522,E2 -13994.522} C_VEL
LIN {X 0,Y 340.745,Z 527.037,A -85,B 0,C 180,E1 -13997.945,E2 -13997.945} C_VEL
LIN {X 0,Y 340.727,Z 527.039,A -85,B 0,C 180,E1 -14000.252,E2 -14000.252} C_VEL
LIN {X 0,Y 340.703,Z 527.044,A -85,B 0,C 180,E1 -14003.559,E2 -14003.559} C_VEL
LIN {X 0,Y 340.685,Z 527.044,A -85,B 0,C 180,E1 -14006.153,E2 -14006.153} C_VEL
LIN {X 0,Y 340.767,Z 527.034,A -85,B 0,C 180,E1 -14010.332,E2 -14010.332} C_VEL
LIN {X 0,Y 340.797,Z 527.036,A -85,B 0,C 180,E1 -14013.02,E2 -14013.02} C_VEL
LIN {X 0,Y 340.746,Z 527.038,A -85,B 0,C 180,E1 -14015.638,E2 -14015.638} C_VEL
LIN {X 0,Y 340.726,Z 527.042,A -85,B 0,C 180,E1 -14019.474,E2 -14019.474} C_VEL
LIN {X 0,Y 340.849,Z 527.024,A -85,B 0,C 180,E1 -14021.984,E2 -14021.984} C_VEL
LIN {X 0,Y 340.861,Z 527.024,A -85,B 0,C 180,E1 -14025.705,E2 -14025.705} C_VEL
LIN {X 0,Y 340.867,Z 527.026,A -85,B 0,C 180,E1 -14029.307,E2 -14029.307} C_VEL
LIN {X 0,Y 341.07,Z 527,A -85,B 0,C 180,E1 -14032.899,E2 -14032.899} C_VEL
LIN {X 0,Y 341.163,Z 526.987,A -85,B 0,C 180,E1 -14037.639,E2 -14037.639} C_VEL
LIN {X 0,Y 341.309,Z 526.967,A -85,B 0,C 180,E1 -14040.001,E2 -14040.001} C_VEL
LIN {X 0,Y 341.171,Z 526.984,A -85,B 0,C 180,E1 -14042.362,E2 -14042.362} C_VEL
LIN {X 0,Y 341.055,Z 527.003,A -85,B 0,C 180,E1 -14047.103,E2 -14047.103} C_VEL
LIN {X 0,Y 340.864,Z 527.023,A -85,B 0,C 180,E1 -14050.695,E2 -14050.695} C_VEL
LIN {X 0,Y 340.857,Z 527.023,A -85,B 0,C 180,E1 -14054.326,E2 -14054.326} C_VEL
LIN {X 0,Y 340.831,Z 527.026,A -85,B 0,C 180,E1 -14058.467,E2 -14058.467} C_VEL
LIN {X 0,Y 340.748,Z 527.037,A -85,B 0,C 180,E1 -14061.858,E2 -14061.858} C_VEL
LIN {X 0,Y 340.768,Z 527.036,A -85,B 0,C 180,E1 -14065.665,E2 -14065.665} C_VEL
LIN {X 0,Y 340.738,Z 527.038,A -85,B 0,C 180,E1 -14068.321,E2 -14068.321} C_VEL
LIN {X 0,Y 340.712,Z 527.044,A -85,B 0,C 180,E1 -14071.044,E2 -14071.044} C_VEL
LIN {X 0,Y 340.715,Z 527.047,A -85,B 0,C 180,E1 -14075.28,E2 -14075.28} C_VEL
LIN {X 0,Y 340.709,Z 527.041,A -85,B 0,C 180,E1 -14078.388,E2 -14078.388} C_VEL
LIN {X 0,Y 340.697,Z 527.043,A -85,B 0,C 180,E1 -14082.047,E2 -14082.047} C_VEL
LIN {X 0,Y 340.719,Z 527.045,A -85,B 0,C 180,E1 -14085.469,E2 -14085.469} C_VEL
LIN {X 0,Y 340.724,Z 527.04,A -85,B 0,C 180,E1 -14088.697,E2 -14088.697} C_VEL
LIN {X 0,Y 340.739,Z 527.04,A -85,B 0,C 180,E1 -14091.775,E2 -14091.775} C_VEL
LIN {X 0,Y 340.723,Z 527.045,A -85,B 0,C 180,E1 -14095.596,E2 -14095.596} C_VEL
LIN {X 0,Y 340.746,Z 527.239,A -85,B 0,C 180,E1 -14097.741,E2 -14097.741} C_VEL
LIN {X 0,Y 343.561,Z 540.107,A -85,B 0,C 180,E1 -14101.125,E2 -14101.125} C_VEL
LIN {X 0,Y 345.29,Z 549.127,A -85,B 0,C 180,E1 -14103.399,E2 -14103.399} C_VEL
LIN {X 0,Y 344.204,Z 560.031,A -85,B 0,C 180,E1 -14105.899,E2 -14105.899} C_VEL
LIN {X 0,Y 343.696,Z 564.835,A -85,B 0,C 180,E1 -14106.99,E2 -14106.99} C_VEL
LIN {X 0,Y 349.162,Z 604.182,A -85,B 0,C 180,E1 -14108.245,E2 -14108.245} C_VEL
LIN {X 0,Y 347.747,Z 674.114,A -85,B 0,C 180,E1 -14109.79,E2 -14109.79} C_VEL
LIN {X 0,Y 346.922,Z 687.745,A -85,B 0,C 180,E1 -14110.319,E2 -14110.319} C_VEL
LIN {X 0,Y 345.979,Z 700.143,A -85,B 0,C 180,E1 -14111.034,E2 -14111.034} C_VEL
LIN {X 0,Y 345.02,Z 711.276,A -85,B 0,C 180,E1 -14111.903,E2 -14111.903} C_VEL
LIN {X 0,Y 343.818,Z 722.893,A -85,B 0,C 180,E1 -14113.066,E2 -14113.066} C_VEL
LIN {X 0,Y 342.723,Z 733.383,A -85,B 0,C 180,E1 -14114.387,E2 -14114.387} C_VEL
LIN {X 0,Y 341.625,Z 743.637,A -85,B 0,C 180,E1 -14116.012,E2 -14116.012} C_VEL
LIN {X 0,Y 340.644,Z 752.619,A -85,B 0,C 180,E1 -14117.792,E2 -14117.792} C_VEL
LIN {X 0,Y 339.937,Z 759.818,A -85,B 0,C 180,E1 -14119.578,E2 -14119.578} C_VEL
LIN {X 0,Y 339.44,Z 766.367,A -85,B 0,C 180,E1 -14121.667,E2 -14121.667} C_VEL
LIN {X 0,Y 339.237,Z 770.8,A -85,B 0,C 180,E1 -14123.517,E2 -14123.517} C_VEL
LIN {X 0,Y 339.174,Z 773.882,A -85,B 0,C 180,E1 -14125.246,E2 -14125.246} C_VEL
LIN {X 0,Y 339.148,Z 775.466,A -85,B 0,C 180,E1 -14126.436,E2 -14126.436} C_VEL
LIN {X 0,Y 339.196,Z 776.617,A -85,B 0,C 180,E1 -14127.625,E2 -14127.625} C_VEL
LIN {X 0,Y 339.304,Z 777.322,A -85,B 0,C 180,E1 -14128.813,E2 -14128.813} C_VEL
LIN {X 0,Y 339.324,Z 777.621,A -85,B 0,C 180,E1 -14130,E2 -14130} C_VEL
LIN {X 0,Y 339.3,Z 777.518,A -85,B 0,C 180,E1 -14131.187,E2 -14131.187} C_VEL
LIN {X 0,Y 339.17,Z 776.992,A -85,B 0,C 180,E1 -14132.375,E2 -14132.375} C_VEL
LIN {X 0,Y 339.132,Z 776.031,A -85,B 0,C 180,E1 -14133.564,E2 -14133.564} C_VEL
LIN {X 0,Y 339.145,Z 774.668,A -85,B 0,C 180,E1 -14134.755,E2 -14134.755} C_VEL
LIN {X 0,Y 339.204,Z 771.806,A -85,B 0,C 180,E1 -14136.543,E2 -14136.543} C_VEL
LIN {X 0,Y 339.436,Z 767.907,A -85,B 0,C 180,E1 -14138.333,E2 -14138.333} C_VEL
LIN {X 0,Y 339.858,Z 762.878,A -85,B 0,C 180,E1 -14140.123,E2 -14140.123} C_VEL
LIN {X 0,Y 340.528,Z 756.579,A -85,B 0,C 180,E1 -14141.91,E2 -14141.91} C_VEL
LIN {X 0,Y 341.597,Z 748.778,A -85,B 0,C 180,E1 -14143.686,E2 -14143.686} C_VEL
LIN {X 0,Y 342.806,Z 739.008,A -85,B 0,C 180,E1 -14145.457,E2 -14145.457} C_VEL
LIN {X 0,Y 344.112,Z 728.966,A -85,B 0,C 180,E1 -14146.92,E2 -14146.92} C_VEL
LIN {X 0,Y 345.521,Z 717.696,A -85,B 0,C 180,E1 -14148.224,E2 -14148.224} C_VEL
LIN {X 0,Y 346.754,Z 706.708,A -85,B 0,C 180,E1 -14149.229,E2 -14149.229} C_VEL
LIN {X 0,Y 347.949,Z 694.631,A -85,B 0,C 180,E1 -14150.082,E2 -14150.082} C_VEL
LIN {X 0,Y 348.974,Z 682.298,A -85,B 0,C 180,E1 -14150.713,E2 -14150.713} C_VEL
LIN {X 0,Y 349.748,Z 668.424,A -85,B 0,C 180,E1 -14151.166,E2 -14151.166} C_VEL
LIN {X 0,Y 351.105,Z 604.111,A -85,B 0,C 180,E1 -14152.6,E2 -14152.6} C_VEL
LIN {X 0,Y 347.715,Z 579.435,A -85,B 0,C 180,E1 -14153.467,E2 -14153.467} C_VEL
LIN {X 0,Y 344.657,Z 562.844,A -85,B 0,C 180,E1 -14154.148,E2 -14154.148} C_VEL
LIN {X 0,Y 345.999,Z 551.274,A -85,B 0,C 180,E1 -14156.867,E2 -14156.867} C_VEL
LIN {X 0,Y 344.26,Z 542.05,A -85,B 0,C 180,E1 -14159.337,E2 -14159.337} C_VEL
LIN {X 0,Y 341.671,Z 530.985,A -85,B 0,C 180,E1 -14162.504,E2 -14162.504} C_VEL
LIN {X 0,Y 340.727,Z 527.05,A -85,B 0,C 180,E1 -14163.753,E2 -14163.753} C_VEL
LIN {X 0,Y 340.706,Z 527.049,A -85,B 0,C 180,E1 -14166.74,E2 -14166.74} C_VEL
LIN {X 0,Y 340.763,Z 527.04,A -85,B 0,C 180,E1 -14170.261,E2 -14170.261} C_VEL
LIN {X 0,Y 340.717,Z 527.043,A -85,B 0,C 180,E1 -14173.784,E2 -14173.784} C_VEL
LIN {X 0,Y 340.677,Z 527.046,A -85,B 0,C 180,E1 -14177.095,E2 -14177.095} C_VEL
LIN {X 0,Y 340.696,Z 527.043,A -85,B 0,C 180,E1 -14180.246,E2 -14180.246} C_VEL
LIN {X 0,Y 340.708,Z 527.042,A -85,B 0,C 180,E1 -14183.558,E2 -14183.558} C_VEL
LIN {X 0,Y 340.688,Z 527.042,A -85,B 0,C 180,E1 -14186.152,E2 -14186.152} C_VEL
LIN {X 0,Y 340.771,Z 527.036,A -85,B 0,C 180,E1 -14190.331,E2 -14190.331} C_VEL
LIN {X 0,Y 340.8,Z 527.031,A -85,B 0,C 180,E1 -14193.019,E2 -14193.019} C_VEL
LIN {X 0,Y 340.723,Z 527.042,A -85,B 0,C 180,E1 -14196.926,E2 -14196.926} C_VEL
LIN {X 0,Y 340.784,Z 527.035,A -85,B 0,C 180,E1 -14200.733,E2 -14200.733} C_VEL
LIN {X 0,Y 340.78,Z 527.032,A -85,B 0,C 180,E1 -14203.218,E2 -14203.218} C_VEL
LIN {X 0,Y 340.837,Z 527.024,A -85,B 0,C 180,E1 -14206.89,E2 -14206.89} C_VEL
LIN {X 0,Y 340.919,Z 527.012,A -85,B 0,C 180,E1 -14210.507,E2 -14210.507} C_VEL
LIN {X 0,Y 341.057,Z 526.999,A -85,B 0,C 180,E1 -14212.897,E2 -14212.897} C_VEL
LIN {X 0,Y 341.163,Z 526.985,A -85,B 0,C 180,E1 -14217.638,E2 -14217.638} C_VEL
LIN {X 0,Y 341.309,Z 526.966,A -85,B 0,C 180,E1 -14219.999,E2 -14219.999} C_VEL
LIN {X 0,Y 341.163,Z 526.988,A -85,B 0,C 180,E1 -14222.361,E2 -14222.361} C_VEL
LIN {X 0,Y 341.054,Z 527.001,A -85,B 0,C 180,E1 -14227.102,E2 -14227.102} C_VEL
LIN {X 0,Y 340.863,Z 527.027,A -85,B 0,C 180,E1 -14230.693,E2 -14230.693} C_VEL
LIN {X 0,Y 340.855,Z 527.026,A -85,B 0,C 180,E1 -14234.325,E2 -14234.325} C_VEL
LIN {X 0,Y 340.829,Z 527.031,A -85,B 0,C 180,E1 -14238.466,E2 -14238.466} C_VEL
LIN {X 0,Y 340.746,Z 527.042,A -85,B 0,C 180,E1 -14241.857,E2 -14241.857} C_VEL
LIN {X 0,Y 340.762,Z 527.044,A -85,B 0,C 180,E1 -14245.664,E2 -14245.664} C_VEL
LIN {X 0,Y 340.788,Z 527.091,A -85,B 0,C 180,E1 -14246.402,E2 -14246.402} C_VEL
LIN {X 0,Y 341.581,Z 530.658,A -85,B 0,C 180,E1 -14247.681,E2 -14247.681} C_VEL
LIN {X 0,Y 349.482,Z 548.666,A -85,B 0,C 180,E1 -14248.816,E2 -14248.816} C_VEL
LIN {X 0,Y 352.177,Z 555.549,A -85,B 0,C 180,E1 -14249.203,E2 -14249.203} C_VEL
LIN {X 0,Y 350.096,Z 637.031,A -85,B 0,C 180,E1 -14251.038,E2 -14251.038} C_VEL
LIN {X 0,Y 349.426,Z 650.638,A -85,B 0,C 180,E1 -14251.59,E2 -14251.59} C_VEL
LIN {X 0,Y 348.749,Z 662.306,A -85,B 0,C 180,E1 -14252.289,E2 -14252.289} C_VEL
LIN {X 0,Y 347.671,Z 674.456,A -85,B 0,C 180,E1 -14253.257,E2 -14253.257} C_VEL
LIN {X 0,Y 346.52,Z 685.595,A -85,B 0,C 180,E1 -14254.405,E2 -14254.405} C_VEL
LIN {X 0,Y 345.338,Z 695.105,A -85,B 0,C 180,E1 -14255.619,E2 -14255.619} C_VEL
LIN {X 0,Y 343.97,Z 704.925,A -85,B 0,C 180,E1 -14257.172,E2 -14257.172} C_VEL
LIN {X 0,Y 342.833,Z 713.305,A -85,B 0,C 180,E1 -14258.833,E2 -14258.833} C_VEL
LIN {X 0,Y 341.812,Z 720.023,A -85,B 0,C 180,E1 -14260.471,E2 -14260.471} C_VEL
LIN {X 0,Y 341.034,Z 725.457,A -85,B 0,C 180,E1 -14262.109,E2 -14262.109} C_VEL
LIN {X 0,Y 340.418,Z 729.783,A -85,B 0,C 180,E1 -14263.733,E2 -14263.733} C_VEL
LIN {X 0,Y 339.975,Z 733.157,A -85,B 0,C 180,E1 -14265.345,E2 -14265.345} C_VEL
LIN {X 0,Y 339.575,Z 735.664,A -85,B 0,C 180,E1 -14266.924,E2 -14266.924} C_VEL
LIN {X 0,Y 339.319,Z 737.358,A -85,B 0,C 180,E1 -14268.489,E2 -14268.489} C_VEL
LIN {X 0,Y 339.144,Z 738.374,A -85,B 0,C 180,E1 -14270.061,E2 -14270.061} C_VEL
LIN {X 0,Y 339.02,Z 738.66,A -85,B 0,C 180,E1 -14271.975,E2 -14271.975} C_VEL
LIN {X 0,Y 339.081,Z 737.874,A -85,B 0,C 180,E1 -14273.933,E2 -14273.933} C_VEL
LIN {X 0,Y 339.27,Z 735.86,A -85,B 0,C 180,E1 -14275.993,E2 -14275.993} C_VEL
LIN {X 0,Y 339.656,Z 732.619,A -85,B 0,C 180,E1 -14278.032,E2 -14278.032} C_VEL
LIN {X 0,Y 340.186,Z 727.448,A -85,B 0,C 180,E1 -14280.277,E2 -14280.277} C_VEL
LIN {X 0,Y 340.852,Z 721.868,A -85,B 0,C 180,E1 -14282.097,E2 -14282.097} C_VEL
LIN {X 0,Y 341.761,Z 714.11,A -85,B 0,C 180,E1 -14284.089,E2 -14284.089} C_VEL
LIN {X 0,Y 342.703,Z 705.717,A -85,B 0,C 180,E1 -14285.786,E2 -14285.786} C_VEL
LIN {X 0,Y 343.724,Z 696.488,A -85,B 0,C 180,E1 -14287.299,E2 -14287.299} C_VEL
LIN {X 0,Y 344.801,Z 685.757,A -85,B 0,C 180,E1 -14288.719,E2 -14288.719} C_VEL
LIN {X 0,Y 345.946,Z 673.817,A -85,B 0,C 180,E1 -14289.952,E2 -14289.952} C_VEL
LIN {X 0,Y 346.841,Z 661.66,A -85,B 0,C 180,E1 -14290.93,E2 -14290.93} C_VEL
LIN {X 0,Y 347.558,Z 648.529,A -85,B 0,C 180,E1 -14291.7,E2 -14291.7} C_VEL
LIN {X 0,Y 348.105,Z 634.73,A -85,B 0,C 180,E1 -14292.241,E2 -14292.241} C_VEL
LIN {X 0,Y 349.933,Z 553.779,A -85,B 0,C 180,E1 -14294.007,E2 -14294.007} C_VEL
LIN {X 0,Y 345.714,Z 540.949,A -85,B 0,C 180,E1 -14294.563,E2 -14294.563} C_VEL
LIN {X 0,Y 341.079,Z 528.25,A -85,B 0,C 180,E1 -14295.19,E2 -14295.19} C_VEL
LIN {X 0,Y 340.882,Z 527.02,A -85,B 0,C 180,E1 -14295.6,E2 -14295.6} C_VEL
LIN {X 0,Y 340.868,Z 527.024,A -85,B 0,C 180,E1 -14299.306,E2 -14299.306} C_VEL
LIN {X 0,Y 341.057,Z 527.004,A -85,B 0,C 180,E1 -14302.898,E2 -14302.898} C_VEL
LIN {X 0,Y 341.167,Z 526.985,A -85,B 0,C 180,E1 -14307.639,E2 -14307.639} C_VEL
LIN {X 0,Y 341.294,Z 526.968,A -85,B 0,C 180,E1 -14310,E2 -14310} C_VEL
LIN {X 0,Y 341.167,Z 526.985,A -85,B 0,C 180,E1 -14312.361,E2 -14312.361} C_VEL
LIN {X 0,Y 341.073,Z 527,A -85,B 0,C 180,E1 -14317.102,E2 -14317.102} C_VEL
LIN {X 0,Y 340.868,Z 527.025,A -85,B 0,C 180,E1 -14320.694,E2 -14320.694} C_VEL
LIN {X 0,Y 340.859,Z 527.023,A -85,B 0,C 180,E1 -14324.325,E2 -14324.325} C_VEL
LIN {X 0,Y 340.833,Z 527.027,A -85,B 0,C 180,E1 -14328.466,E2 -14328.466} C_VEL
LIN {X 0,Y 340.749,Z 527.036,A -85,B 0,C 180,E1 -14331.857,E2 -14331.857} C_VEL
LIN {X 0,Y 340.766,Z 527.035,A -85,B 0,C 180,E1 -14335.718,E2 -14335.718} C_VEL
LIN {X 0,Y 340.081,Z 527.124,A -85,B 0,C 180,E1 -14336.704,E2 -14336.704} C_VEL
LIN {X 0,Y 337.225,Z 527.476,A -85,B 0,C 180,E1 -14338.31,E2 -14338.31} C_VEL
LIN {X 0,Y 334.802,Z 527.778,A -85,B 0,C 180,E1 -14339.609,E2 -14339.609} C_VEL
LIN {X 0,Y 333.743,Z 527.911,A -85,B 0,C 180,E1 -14340.615,E2 -14340.615} C_VEL
LIN {X 0,Y 333.647,Z 527.919,A -85,B 0,C 180,E1 -14340.956,E2 -14340.956} C_VEL
LIN {X 0,Y 333.68,Z 527.92,A -85,B 0,C 180,E1 -14344.774,E2 -14344.774} C_VEL
LIN {X 0,Y 333.677,Z 527.921,A -85,B 0,C 180,E1 -14348.804,E2 -14348.804} C_VEL
LIN {X 0,Y 333.697,Z 527.916,A -85,B 0,C 180,E1 -14352.513,E2 -14352.513} C_VEL
LIN {X 0,Y 333.722,Z 527.912,A -85,B 0,C 180,E1 -14355.977,E2 -14355.977} C_VEL
LIN {X 0,Y 333.695,Z 527.919,A -85,B 0,C 180,E1 -14359.304,E2 -14359.304} C_VEL
LIN {X 0,Y 333.659,Z 527.925,A -85,B 0,C 180,E1 -14363.167,E2 -14363.167} C_VEL
LIN {X 0,Y 333.629,Z 527.926,A -85,B 0,C 180,E1 -14366.792,E2 -14366.792} C_VEL
LIN {X 0,Y 333.695,Z 527.916,A -85,B 0,C 180,E1 -14369.71,E2 -14369.71} C_VEL
LIN {X 0,Y 333.736,Z 527.91,A -85,B 0,C 180,E1 -14372.401,E2 -14372.401} C_VEL
LIN {X 0,Y 333.718,Z 527.918,A -85,B 0,C 180,E1 -14375.091,E2 -14375.091} C_VEL
LIN {X 0,Y 333.665,Z 527.923,A -85,B 0,C 180,E1 -14379.019,E2 -14379.019} C_VEL
LIN {X 0,Y 333.785,Z 527.906,A -85,B 0,C 180,E1 -14381.59,E2 -14381.59} C_VEL
LIN {X 0,Y 333.8,Z 527.904,A -85,B 0,C 180,E1 -14385.577,E2 -14385.577} C_VEL
LIN {X 0,Y 333.829,Z 527.903,A -85,B 0,C 180,E1 -14389.079,E2 -14389.079} C_VEL
LIN {X 0,Y 334.019,Z 527.876,A -85,B 0,C 180,E1 -14392.748,E2 -14392.748} C_VEL
LIN {X 0,Y 333.81,Z 527.907,A -85,B 0,C 180,E1 -14395.17,E2 -14395.17} C_VEL
LIN {X 0,Y 334.1,Z 527.867,A -85,B 0,C 180,E1 -14397.589,E2 -14397.589} C_VEL
LIN {X 0,Y 334.26,Z 527.845,A -85,B 0,C 180,E1 -14400.001,E2 -14400.001} C_VEL
LIN {X 0,Y 334.133,Z 527.86,A -85,B 0,C 180,E1 -14402.412,E2 -14402.412} C_VEL
LIN {X 0,Y 334.012,Z 527.876,A -85,B 0,C 180,E1 -14406.04,E2 -14406.04} C_VEL
LIN {X 0,Y 333.952,Z 527.883,A -85,B 0,C 180,E1 -14408.472,E2 -14408.472} C_VEL
LIN {X 0,Y 333.784,Z 527.904,A -85,B 0,C 180,E1 -14412.155,E2 -14412.155} C_VEL
LIN {X 0,Y 333.771,Z 527.906,A -85,B 0,C 180,E1 -14415.887,E2 -14415.887} C_VEL
LIN {X 0,Y 333.79,Z 527.904,A -85,B 0,C 180,E1 -14418.656,E2 -14418.656} C_VEL
LIN {X 0,Y 333.687,Z 527.916,A -85,B 0,C 180,E1 -14422.279,E2 -14422.279} C_VEL
LIN {X 0,Y 333.731,Z 527.911,A -85,B 0,C 180,E1 -14426.247,E2 -14426.247} C_VEL
LIN {X 0,Y 333.707,Z 527.916,A -85,B 0,C 180,E1 -14428.973,E2 -14428.973} C_VEL
LIN {X 0,Y 333.647,Z 527.921,A -85,B 0,C 180,E1 -14432.59,E2 -14432.59} C_VEL
LIN {X 0,Y 333.674,Z 527.918,A -85,B 0,C 180,E1 -14436.14,E2 -14436.14} C_VEL
LIN {X 0,Y 333.644,Z 527.926,A -85,B 0,C 180,E1 -14439.193,E2 -14439.193} C_VEL
LIN {X 0,Y 333.632,Z 527.923,A -85,B 0,C 180,E1 -14442.501,E2 -14442.501} C_VEL
LIN {X 0,Y 333.665,Z 527.92,A -85,B 0,C 180,E1 -14445.968,E2 -14445.968} C_VEL
LIN {X 0,Y 333.701,Z 527.92,A -85,B 0,C 180,E1 -14449.306,E2 -14449.306} C_VEL
LIN {X 0,Y 333.666,Z 527.923,A -85,B 0,C 180,E1 -14453.169,E2 -14453.169} C_VEL
LIN {X 0,Y 333.645,Z 527.927,A -85,B 0,C 180,E1 -14456.793,E2 -14456.793} C_VEL
LIN {X 0,Y 333.668,Z 527.972,A -85,B 0,C 180,E1 -14457.338,E2 -14457.338} C_VEL
LIN {X 0,Y 336.328,Z 540.009,A -85,B 0,C 180,E1 -14460.591,E2 -14460.591} C_VEL
LIN {X 0,Y 338.336,Z 550.435,A -85,B 0,C 180,E1 -14463.28,E2 -14463.28} C_VEL
LIN {X 0,Y 336.89,Z 564.23,A -85,B 0,C 180,E1 -14466.503,E2 -14466.503} C_VEL
LIN {X 0,Y 336.869,Z 564.506,A -85,B 0,C 180,E1 -14466.567,E2 -14466.567} C_VEL
LIN {X 0,Y 342.446,Z 605.14,A -85,B 0,C 180,E1 -14467.879,E2 -14467.879} C_VEL
LIN {X 0,Y 341.01,Z 673.347,A -85,B 0,C 180,E1 -14469.415,E2 -14469.415} C_VEL
LIN {X 0,Y 340.216,Z 687.045,A -85,B 0,C 180,E1 -14469.954,E2 -14469.954} C_VEL
LIN {X 0,Y 339.286,Z 698.967,A -85,B 0,C 180,E1 -14470.645,E2 -14470.645} C_VEL
LIN {X 0,Y 338.235,Z 710.314,A -85,B 0,C 180,E1 -14471.527,E2 -14471.527} C_VEL
LIN {X 0,Y 337.005,Z 722.044,A -85,B 0,C 180,E1 -14472.713,E2 -14472.713} C_VEL
LIN {X 0,Y 335.842,Z 732.609,A -85,B 0,C 180,E1 -14474.059,E2 -14474.059} C_VEL
LIN {X 0,Y 334.927,Z 741.257,A -85,B 0,C 180,E1 -14475.416,E2 -14475.416} C_VEL
LIN {X 0,Y 334.005,Z 749.22,A -85,B 0,C 180,E1 -14476.927,E2 -14476.927} C_VEL
LIN {X 0,Y 333.086,Z 756.975,A -85,B 0,C 180,E1 -14478.746,E2 -14478.746} C_VEL
LIN {X 0,Y 332.508,Z 764.13,A -85,B 0,C 180,E1 -14480.879,E2 -14480.879} C_VEL
LIN {X 0,Y 332.234,Z 768.866,A -85,B 0,C 180,E1 -14482.708,E2 -14482.708} C_VEL
LIN {X 0,Y 332.141,Z 771.499,A -85,B 0,C 180,E1 -14483.996,E2 -14483.996} C_VEL
LIN {X 0,Y 332.09,Z 773.403,A -85,B 0,C 180,E1 -14485.144,E2 -14485.144} C_VEL
LIN {X 0,Y 332.071,Z 775.001,A -85,B 0,C 180,E1 -14486.36,E2 -14486.36} C_VEL
LIN {X 0,Y 332.101,Z 776.174,A -85,B 0,C 180,E1 -14487.574,E2 -14487.574} C_VEL
LIN {X 0,Y 332.209,Z 776.893,A -85,B 0,C 180,E1 -14488.788,E2 -14488.788} C_VEL
LIN {X 0,Y 332.265,Z 777.205,A -85,B 0,C 180,E1 -14490,E2 -14490} C_VEL
LIN {X 0,Y 332.204,Z 777.111,A -85,B 0,C 180,E1 -14491.212,E2 -14491.212} C_VEL
LIN {X 0,Y 332.075,Z 776.605,A -85,B 0,C 180,E1 -14492.426,E2 -14492.426} C_VEL
LIN {X 0,Y 332.056,Z 775.657,A -85,B 0,C 180,E1 -14493.64,E2 -14493.64} C_VEL
LIN {X 0,Y 332.078,Z 772.81,A -85,B 0,C 180,E1 -14495.901,E2 -14495.901} C_VEL
LIN {X 0,Y 332.27,Z 769.024,A -85,B 0,C 180,E1 -14497.902,E2 -14497.902} C_VEL
LIN {X 0,Y 332.665,Z 764.42,A -85,B 0,C 180,E1 -14499.73,E2 -14499.73} C_VEL
LIN {X 0,Y 333.391,Z 757.485,A -85,B 0,C 180,E1 -14501.86,E2 -14501.86} C_VEL
LIN {X 0,Y 334.497,Z 749.971,A -85,B 0,C 180,E1 -14503.672,E2 -14503.672} C_VEL
LIN {X 0,Y 335.728,Z 740.765,A -85,B 0,C 180,E1 -14505.463,E2 -14505.463} C_VEL
LIN {X 0,Y 337.012,Z 731.043,A -85,B 0,C 180,E1 -14506.975,E2 -14506.975} C_VEL
LIN {X 0,Y 338.439,Z 720.407,A -85,B 0,C 180,E1 -14508.305,E2 -14508.305} C_VEL
LIN {X 0,Y 339.883,Z 708.617,A -85,B 0,C 180,E1 -14509.476,E2 -14509.476} C_VEL
LIN {X 0,Y 341.245,Z 696.095,A -85,B 0,C 180,E1 -14510.415,E2 -14510.415} C_VEL
LIN {X 0,Y 342.365,Z 683.032,A -85,B 0,C 180,E1 -14511.132,E2 -14511.132} C_VEL
LIN {X 0,Y 343.154,Z 670.148,A -85,B 0,C 180,E1 -14511.592,E2 -14511.592} C_VEL
LIN {X 0,Y 344.68,Z 604.969,A -85,B 0,C 180,E1 -14513.081,E2 -14513.081} C_VEL
LIN {X 0,Y 341.815,Z 583.631,A -85,B 0,C 180,E1 -14513.848,E2 -14513.848} C_VEL
LIN {X 0,Y 338.368,Z 564.615,A -85,B 0,C 180,E1 -14514.631,E2 -14514.631} C_VEL
LIN {X 0,Y 337.931,Z 562.378,A -85,B 0,C 180,E1 -14514.742,E2 -14514.742} C_VEL
LIN {X 0,Y 339.152,Z 553.026,A -85,B 0,C 180,E1 -14516.993,E2 -14516.993} C_VEL
LIN {X 0,Y 337.484,Z 544.097,A -85,B 0,C 180,E1 -14519.435,E2 -14519.435} C_VEL
LIN {X 0,Y 335.251,Z 534.353,A -85,B 0,C 180,E1 -14522.281,E2 -14522.281} C_VEL
LIN {X 0,Y 333.691,Z 527.924,A -85,B 0,C 180,E1 -14524.29,E2 -14524.29} C_VEL
LIN {X 0,Y 333.655,Z 527.924,A -85,B 0,C 180,E1 -14527.65,E2 -14527.65} C_VEL
LIN {X 0,Y 333.698,Z 527.917,A -85,B 0,C 180,E1 -14530.759,E2 -14530.759} C_VEL
LIN {X 0,Y 333.678,Z 527.922,A -85,B 0,C 180,E1 -14534.265,E2 -14534.265} C_VEL
LIN {X 0,Y 333.641,Z 527.92,A -85,B 0,C 180,E1 -14537.618,E2 -14537.618} C_VEL
LIN {X 0,Y 333.651,Z 527.925,A -85,B 0,C 180,E1 -14541.201,E2 -14541.201} C_VEL
LIN {X 0,Y 333.674,Z 527.918,A -85,B 0,C 180,E1 -14543.86,E2 -14543.86} C_VEL
LIN {X 0,Y 333.639,Z 527.925,A -85,B 0,C 180,E1 -14547.412,E2 -14547.412} C_VEL
LIN {X 0,Y 333.707,Z 527.917,A -85,B 0,C 180,E1 -14551.027,E2 -14551.027} C_VEL
LIN {X 0,Y 333.731,Z 527.913,A -85,B 0,C 180,E1 -14553.753,E2 -14553.753} C_VEL
LIN {X 0,Y 333.714,Z 527.914,A -85,B 0,C 180,E1 -14557.913,E2 -14557.913} C_VEL
LIN {X 0,Y 333.787,Z 527.905,A -85,B 0,C 180,E1 -14561.588,E2 -14561.588} C_VEL
LIN {X 0,Y 333.802,Z 527.901,A -85,B 0,C 180,E1 -14565.576,E2 -14565.576} C_VEL
LIN {X 0,Y 333.827,Z 527.9,A -85,B 0,C 180,E1 -14569.077,E2 -14569.077} C_VEL
LIN {X 0,Y 334.008,Z 527.879,A -85,B 0,C 180,E1 -14572.747,E2 -14572.747} C_VEL
LIN {X 0,Y 333.809,Z 527.906,A -85,B 0,C 180,E1 -14575.168,E2 -14575.168} C_VEL
LIN {X 0,Y 334.1,Z 527.865,A -85,B 0,C 180,E1 -14577.588,E2 -14577.588} C_VEL
LIN {X 0,Y 334.26,Z 527.844,A -85,B 0,C 180,E1 -14579.999,E2 -14579.999} C_VEL
LIN {X 0,Y 334.125,Z 527.865,A -85,B 0,C 180,E1 -14582.41,E2 -14582.41} C_VEL
LIN {X 0,Y 333.988,Z 527.878,A -85,B 0,C 180,E1 -14586.596,E2 -14586.596} C_VEL
LIN {X 0,Y 333.843,Z 527.901,A -85,B 0,C 180,E1 -14589.695,E2 -14589.695} C_VEL
LIN {X 0,Y 333.788,Z 527.906,A -85,B 0,C 180,E1 -14593.391,E2 -14593.391} C_VEL
LIN {X 0,Y 333.738,Z 527.914,A -85,B 0,C 180,E1 -14597.146,E2 -14597.146} C_VEL
LIN {X 0,Y 333.73,Z 527.916,A -85,B 0,C 180,E1 -14599.69,E2 -14599.69} C_VEL
LIN {X 0,Y 333.684,Z 527.922,A -85,B 0,C 180,E1 -14602.278,E2 -14602.278} C_VEL
LIN {X 0,Y 333.752,Z 528.086,A -85,B 0,C 180,E1 -14605.894,E2 -14605.894} C_VEL
LIN {X 0,Y 334.475,Z 531.131,A -85,B 0,C 180,E1 -14607.025,E2 -14607.025} C_VEL
LIN {X 0,Y 342.364,Z 548.7,A -85,B 0,C 180,E1 -14608.214,E2 -14608.214} C_VEL
LIN {X 0,Y 345.85,Z 557.468,A -85,B 0,C 180,E1 -14608.732,E2 -14608.732} C_VEL
LIN {X 0,Y 343.636,Z 637.541,A -85,B 0,C 180,E1 -14610.566,E2 -14610.566} C_VEL
LIN {X 0,Y 342.926,Z 651.391,A -85,B 0,C 180,E1 -14611.141,E2 -14611.141} C_VEL
LIN {X 0,Y 342.124,Z 664.079,A -85,B 0,C 180,E1 -14611.935,E2 -14611.935} C_VEL
LIN {X 0,Y 340.953,Z 676.107,A -85,B 0,C 180,E1 -14612.938,E2 -14612.938} C_VEL
LIN {X 0,Y 339.649,Z 687.951,A -85,B 0,C 180,E1 -14614.222,E2 -14614.222} C_VEL
LIN {X 0,Y 338.324,Z 697.771,A -85,B 0,C 180,E1 -14615.565,E2 -14615.565} C_VEL
LIN {X 0,Y 336.895,Z 707.545,A -85,B 0,C 180,E1 -14617.226,E2 -14617.226} C_VEL
LIN {X 0,Y 335.704,Z 715.489,A -85,B 0,C 180,E1 -14618.906,E2 -14618.906} C_VEL
LIN {X 0,Y 334.538,Z 722.818,A -85,B 0,C 180,E1 -14620.863,E2 -14620.863} C_VEL
LIN {X 0,Y 333.635,Z 728.87,A -85,B 0,C 180,E1 -14622.947,E2 -14622.947} C_VEL
LIN {X 0,Y 332.991,Z 733.332,A -85,B 0,C 180,E1 -14625.007,E2 -14625.007} C_VEL
LIN {X 0,Y 332.564,Z 735.941,A -85,B 0,C 180,E1 -14626.661,E2 -14626.661} C_VEL
LIN {X 0,Y 332.33,Z 737.227,A -85,B 0,C 180,E1 -14627.745,E2 -14627.745} C_VEL
LIN {X 0,Y 332.089,Z 738.656,A -85,B 0,C 180,E1 -14629.628,E2 -14629.628} C_VEL
LIN {X 0,Y 331.942,Z 739.12,A -85,B 0,C 180,E1 -14631.57,E2 -14631.57} C_VEL
LIN {X 0,Y 331.978,Z 738.475,A -85,B 0,C 180,E1 -14633.648,E2 -14633.648} C_VEL
LIN {X 0,Y 332.129,Z 736.776,A -85,B 0,C 180,E1 -14635.613,E2 -14635.613} C_VEL
LIN {X 0,Y 332.52,Z 733.724,A -85,B 0,C 180,E1 -14637.716,E2 -14637.716} C_VEL
LIN {X 0,Y 333.02,Z 729.107,A -85,B 0,C 180,E1 -14639.911,E2 -14639.911} C_VEL
LIN {X 0,Y 333.594,Z 724.299,A -85,B 0,C 180,E1 -14641.633,E2 -14641.633} C_VEL
LIN {X 0,Y 334.338,Z 717.888,A -85,B 0,C 180,E1 -14643.469,E2 -14643.469} C_VEL
LIN {X 0,Y 335.23,Z 710.266,A -85,B 0,C 180,E1 -14645.211,E2 -14645.211} C_VEL
LIN {X 0,Y 336.385,Z 700.739,A -85,B 0,C 180,E1 -14646.957,E2 -14646.957} C_VEL
LIN {X 0,Y 337.499,Z 690.448,A -85,B 0,C 180,E1 -14648.469,E2 -14648.469} C_VEL
LIN {X 0,Y 338.701,Z 678.761,A -85,B 0,C 180,E1 -14649.821,E2 -14649.821} C_VEL
LIN {X 0,Y 339.628,Z 668.005,A -85,B 0,C 180,E1 -14650.806,E2 -14650.806} C_VEL
LIN {X 0,Y 340.395,Z 656.518,A -85,B 0,C 180,E1 -14651.627,E2 -14651.627} C_VEL
LIN {X 0,Y 341.101,Z 643.082,A -85,B 0,C 180,E1 -14652.308,E2 -14652.308} C_VEL
LIN {X 0,Y 341.487,Z 629.918,A -85,B 0,C 180,E1 -14652.734,E2 -14652.734} C_VEL
LIN {X 0,Y 343.2,Z 554.653,A -85,B 0,C 180,E1 -14654.396,E2 -14654.396} C_VEL
LIN {X 0,Y 335.697,Z 533.547,A -85,B 0,C 180,E1 -14655.378,E2 -14655.378} C_VEL
LIN {X 0,Y 333.983,Z 528.712,A -85,B 0,C 180,E1 -14655.626,E2 -14655.626} C_VEL
LIN {X 0,Y 333.819,Z 527.9,A -85,B 0,C 180,E1 -14655.98,E2 -14655.98} C_VEL
LIN {X 0,Y 333.858,Z 527.896,A -85,B 0,C 180,E1 -14660.305,E2 -14660.305} C_VEL
LIN {X 0,Y 334.009,Z 527.881,A -85,B 0,C 180,E1 -14662.747,E2 -14662.747} C_VEL
LIN {X 0,Y 333.808,Z 527.904,A -85,B 0,C 180,E1 -14665.169,E2 -14665.169} C_VEL
LIN {X 0,Y 334.104,Z 527.865,A -85,B 0,C 180,E1 -14667.589,E2 -14667.589} C_VEL
LIN {X 0,Y 334.245,Z 527.847,A -85,B 0,C 180,E1 -14670,E2 -14670} C_VEL
LIN {X 0,Y 334.104,Z 527.866,A -85,B 0,C 180,E1 -14672.411,E2 -14672.411} C_VEL
LIN {X 0,Y 334.023,Z 527.877,A -85,B 0,C 180,E1 -14677.252,E2 -14677.252} C_VEL
LIN {X 0,Y 333.831,Z 527.904,A -85,B 0,C 180,E1 -14680.922,E2 -14680.922} C_VEL
LIN {X 0,Y 333.805,Z 527.904,A -85,B 0,C 180,E1 -14684.634,E2 -14684.634} C_VEL
LIN {X 0,Y 333.792,Z 527.906,A -85,B 0,C 180,E1 -14688.655,E2 -14688.655} C_VEL
LIN {X 0,Y 333.688,Z 527.916,A -85,B 0,C 180,E1 -14692.278,E2 -14692.278} C_VEL
LIN {X 0,Y 333.731,Z 527.911,A -85,B 0,C 180,E1 -14696.246,E2 -14696.246} C_VEL
LIN {X 0,Y 333.707,Z 527.919,A -85,B 0,C 180,E1 -14698.972,E2 -14698.972} C_VEL
LIN {X 0,Y 333.647,Z 527.919,A -85,B 0,C 180,E1 -14700.956,E2 -14700.956} C_VEL
LIN {X 0,Y 332.948,Z 528.009,A -85,B 0,C 180,E1 -14701.963,E2 -14701.963} C_VEL
LIN {X 0,Y 330.082,Z 528.366,A -85,B 0,C 180,E1 -14703.602,E2 -14703.602} C_VEL
LIN {X 0,Y 327.68,Z 528.669,A -85,B 0,C 180,E1 -14704.93,E2 -14704.93} C_VEL
LIN {X 0,Y 326.665,Z 528.791,A -85,B 0,C 180,E1 -14705.958,E2 -14705.958} C_VEL
LIN {X 0,Y 326.589,Z 528.8,A -85,B 0,C 180,E1 -14706.306,E2 -14706.306} C_VEL
LIN {X 0,Y 326.64,Z 528.797,A -85,B 0,C 180,E1 -14709.234,E2 -14709.234} C_VEL
LIN {X 0,Y 326.644,Z 528.799,A -85,B 0,C 180,E1 -14712.986,E2 -14712.986} C_VEL
LIN {X 0,Y 326.651,Z 528.793,A -85,B 0,C 180,E1 -14716.49,E2 -14716.49} C_VEL
LIN {X 0,Y 326.628,Z 528.795,A -85,B 0,C 180,E1 -14719.797,E2 -14719.797} C_VEL
LIN {X 0,Y 326.625,Z 528.8,A -85,B 0,C 180,E1 -14722.953,E2 -14722.953} C_VEL
LIN {X 0,Y 326.599,Z 528.799,A -85,B 0,C 180,E1 -14725.981,E2 -14725.981} C_VEL
LIN {X 0,Y 326.653,Z 528.792,A -85,B 0,C 180,E1 -14730.341,E2 -14730.341} C_VEL
LIN {X 0,Y 326.682,Z 528.79,A -85,B 0,C 180,E1 -14734.516,E2 -14734.516} C_VEL
LIN {X 0,Y 326.611,Z 528.798,A -85,B 0,C 180,E1 -14738.544,E2 -14738.544} C_VEL
LIN {X 0,Y 326.737,Z 528.787,A -85,B 0,C 180,E1 -14741.178,E2 -14741.178} C_VEL
LIN {X 0,Y 326.755,Z 528.783,A -85,B 0,C 180,E1 -14745.434,E2 -14745.434} C_VEL
LIN {X 0,Y 326.765,Z 528.781,A -85,B 0,C 180,E1 -14748.839,E2 -14748.839} C_VEL
LIN {X 0,Y 326.973,Z 528.753,A -85,B 0,C 180,E1 -14752.591,E2 -14752.591} C_VEL
LIN {X 0,Y 326.776,Z 528.781,A -85,B 0,C 180,E1 -14755.065,E2 -14755.065} C_VEL
LIN {X 0,Y 327.041,Z 528.746,A -85,B 0,C 180,E1 -14757.537,E2 -14757.537} C_VEL
LIN {X 0,Y 327.21,Z 528.722,A -85,B 0,C 180,E1 -14760.001,E2 -14760.001} C_VEL
LIN {X 0,Y 327.07,Z 528.74,A -85,B 0,C 180,E1 -14762.464,E2 -14762.464} C_VEL
LIN {X 0,Y 326.986,Z 528.751,A -85,B 0,C 180,E1 -14766.17,E2 -14766.17} C_VEL
LIN {X 0,Y 326.799,Z 528.774,A -85,B 0,C 180,E1 -14769.907,E2 -14769.907} C_VEL
LIN {X 0,Y 326.753,Z 528.782,A -85,B 0,C 180,E1 -14773.686,E2 -14773.686} C_VEL
LIN {X 0,Y 326.693,Z 528.79,A -85,B 0,C 180,E1 -14777.529,E2 -14777.529} C_VEL
LIN {X 0,Y 326.66,Z 528.792,A -85,B 0,C 180,E1 -14780.136,E2 -14780.136} C_VEL
LIN {X 0,Y 326.647,Z 528.793,A -85,B 0,C 180,E1 -14784.13,E2 -14784.13} C_VEL
LIN {X 0,Y 326.681,Z 528.791,A -85,B 0,C 180,E1 -14786.859,E2 -14786.859} C_VEL
LIN {X 0,Y 326.638,Z 528.795,A -85,B 0,C 180,E1 -14790.613,E2 -14790.613} C_VEL
LIN {X 0,Y 326.605,Z 528.799,A -85,B 0,C 180,E1 -14794.02,E2 -14794.02} C_VEL
LIN {X 0,Y 326.626,Z 528.801,A -85,B 0,C 180,E1 -14797.24,E2 -14797.24} C_VEL
LIN {X 0,Y 326.576,Z 528.806,A -85,B 0,C 180,E1 -14801.133,E2 -14801.133} C_VEL
LIN {X 0,Y 326.58,Z 528.802,A -85,B 0,C 180,E1 -14804.754,E2 -14804.754} C_VEL
LIN {X 0,Y 326.621,Z 528.797,A -85,B 0,C 180,E1 -14808.162,E2 -14808.162} C_VEL
LIN {X 0,Y 326.646,Z 528.799,A -85,B 0,C 180,E1 -14811.396,E2 -14811.396} C_VEL
LIN {X 0,Y 326.619,Z 528.798,A -85,B 0,C 180,E1 -14814.852,E2 -14814.852} C_VEL
LIN {X 0,Y 326.638,Z 528.947,A -85,B 0,C 180,E1 -14816.995,E2 -14816.995} C_VEL
LIN {X 0,Y 329.241,Z 540.696,A -85,B 0,C 180,E1 -14820.246,E2 -14820.246} C_VEL
LIN {X 0,Y 331.389,Z 551.806,A -85,B 0,C 180,E1 -14823.179,E2 -14823.179} C_VEL
LIN {X 0,Y 330.042,Z 564.026,A -85,B 0,C 180,E1 -14826.093,E2 -14826.093} C_VEL
LIN {X 0,Y 335.279,Z 601.868,A -85,B 0,C 180,E1 -14827.379,E2 -14827.379} C_VEL
LIN {X 0,Y 335.707,Z 607.024,A -85,B 0,C 180,E1 -14827.53,E2 -14827.53} C_VEL
LIN {X 0,Y 334.243,Z 673.23,A -85,B 0,C 180,E1 -14829.057,E2 -14829.057} C_VEL
LIN {X 0,Y 333.409,Z 686.881,A -85,B 0,C 180,E1 -14829.607,E2 -14829.607} C_VEL
LIN {X 0,Y 332.459,Z 698.741,A -85,B 0,C 180,E1 -14830.312,E2 -14830.312} C_VEL
LIN {X 0,Y 331.296,Z 710.837,A -85,B 0,C 180,E1 -14831.286,E2 -14831.286} C_VEL
LIN {X 0,Y 330.039,Z 722.397,A -85,B 0,C 180,E1 -14832.496,E2 -14832.496} C_VEL
LIN {X 0,Y 328.845,Z 732.84,A -85,B 0,C 180,E1 -14833.869,E2 -14833.869} C_VEL
LIN {X 0,Y 327.807,Z 742.221,A -85,B 0,C 180,E1 -14835.41,E2 -14835.41} C_VEL
LIN {X 0,Y 326.675,Z 751.308,A -85,B 0,C 180,E1 -14837.261,E2 -14837.261} C_VEL
LIN {X 0,Y 325.849,Z 758.62,A -85,B 0,C 180,E1 -14839.122,E2 -14839.122} C_VEL
LIN {X 0,Y 325.447,Z 763.55,A -85,B 0,C 180,E1 -14840.679,E2 -14840.679} C_VEL
LIN {X 0,Y 325.168,Z 768.327,A -85,B 0,C 180,E1 -14842.549,E2 -14842.549} C_VEL
LIN {X 0,Y 325.043,Z 771.313,A -85,B 0,C 180,E1 -14844.048,E2 -14844.048} C_VEL
LIN {X 0,Y 324.997,Z 774.528,A -85,B 0,C 180,E1 -14846.28,E2 -14846.28} C_VEL
LIN {X 0,Y 325.008,Z 775.721,A -85,B 0,C 180,E1 -14847.521,E2 -14847.521} C_VEL
LIN {X 0,Y 325.115,Z 776.461,A -85,B 0,C 180,E1 -14848.761,E2 -14848.761} C_VEL
LIN {X 0,Y 325.187,Z 776.787,A -85,B 0,C 180,E1 -14850,E2 -14850} C_VEL
LIN {X 0,Y 325.107,Z 776.706,A -85,B 0,C 180,E1 -14851.239,E2 -14851.239} C_VEL
LIN {X 0,Y 324.984,Z 776.22,A -85,B 0,C 180,E1 -14852.479,E2 -14852.479} C_VEL
LIN {X 0,Y 324.98,Z 775.294,A -85,B 0,C 180,E1 -14853.72,E2 -14853.72} C_VEL
LIN {X 0,Y 324.975,Z 772.765,A -85,B 0,C 180,E1 -14855.835,E2 -14855.835} C_VEL
LIN {X 0,Y 325.202,Z 768.71,A -85,B 0,C 180,E1 -14858.075,E2 -14858.075} C_VEL
LIN {X 0,Y 325.613,Z 764.134,A -85,B 0,C 180,E1 -14859.943,E2 -14859.943} C_VEL
LIN {X 0,Y 326.417,Z 757.247,A -85,B 0,C 180,E1 -14862.118,E2 -14862.118} C_VEL
LIN {X 0,Y 327.567,Z 749.766,A -85,B 0,C 180,E1 -14863.967,E2 -14863.967} C_VEL
LIN {X 0,Y 328.77,Z 741.29,A -85,B 0,C 180,E1 -14865.672,E2 -14865.672} C_VEL
LIN {X 0,Y 330.213,Z 731.009,A -85,B 0,C 180,E1 -14867.335,E2 -14867.335} C_VEL
LIN {X 0,Y 331.721,Z 720.48,A -85,B 0,C 180,E1 -14868.689,E2 -14868.689} C_VEL
LIN {X 0,Y 333.198,Z 708.836,A -85,B 0,C 180,E1 -14869.884,E2 -14869.884} C_VEL
LIN {X 0,Y 334.609,Z 696.551,A -85,B 0,C 180,E1 -14870.839,E2 -14870.839} C_VEL
LIN {X 0,Y 335.775,Z 683.79,A -85,B 0,C 180,E1 -14871.567,E2 -14871.567} C_VEL
LIN {X 0,Y 336.662,Z 670.573,A -85,B 0,C 180,E1 -14872.071,E2 -14872.071} C_VEL
LIN {X 0,Y 338.263,Z 605.708,A -85,B 0,C 180,E1 -14873.587,E2 -14873.587} C_VEL
LIN {X 0,Y 335.099,Z 582.07,A -85,B 0,C 180,E1 -14874.47,E2 -14874.47} C_VEL
LIN {X 0,Y 331.292,Z 561.966,A -85,B 0,C 180,E1 -14875.356,E2 -14875.356} C_VEL
LIN {X 0,Y 332.179,Z 555.879,A -85,B 0,C 180,E1 -14876.848,E2 -14876.848} C_VEL
LIN {X 0,Y 331.976,Z 552.438,A -85,B 0,C 180,E1 -14877.758,E2 -14877.758} C_VEL
LIN {X 0,Y 329.851,Z 542.008,A -85,B 0,C 180,E1 -14880.753,E2 -14880.753} C_VEL
LIN {X 0,Y 327.055,Z 530.465,A -85,B 0,C 180,E1 -14884.337,E2 -14884.337} C_VEL
LIN {X 0,Y 326.642,Z 528.804,A -85,B 0,C 180,E1 -14884.901,E2 -14884.901} C_VEL
LIN {X 0,Y 326.646,Z 528.797,A -85,B 0,C 180,E1 -14888.604,E2 -14888.604} C_VEL
LIN {X 0,Y 326.621,Z 528.8,A -85,B 0,C 180,E1 -14891.837,E2 -14891.837} C_VEL
LIN {X 0,Y 326.584,Z 528.802,A -85,B 0,C 180,E1 -14895.246,E2 -14895.246} C_VEL
LIN {X 0,Y 326.576,Z 528.808,A -85,B 0,C 180,E1 -14898.867,E2 -14898.867} C_VEL
LIN {X 0,Y 326.626,Z 528.796,A -85,B 0,C 180,E1 -14902.76,E2 -14902.76} C_VEL
LIN {X 0,Y 326.603,Z 528.796,A -85,B 0,C 180,E1 -14905.979,E2 -14905.979} C_VEL
LIN {X 0,Y 326.657,Z 528.794,A -85,B 0,C 180,E1 -14910.34,E2 -14910.34} C_VEL
LIN {X 0,Y 326.685,Z 528.793,A -85,B 0,C 180,E1 -14914.515,E2 -14914.515} C_VEL
LIN {X 0,Y 326.64,Z 528.794,A -85,B 0,C 180,E1 -14918.544,E2 -14918.544} C_VEL
LIN {X 0,Y 326.739,Z 528.785,A -85,B 0,C 180,E1 -14921.177,E2 -14921.177} C_VEL
LIN {X 0,Y 326.757,Z 528.78,A -85,B 0,C 180,E1 -14925.432,E2 -14925.432} C_VEL
LIN {X 0,Y 326.763,Z 528.783,A -85,B 0,C 180,E1 -14928.838,E2 -14928.838} C_VEL
LIN {X 0,Y 326.962,Z 528.758,A -85,B 0,C 180,E1 -14932.589,E2 -14932.589} C_VEL
LIN {X 0,Y 326.775,Z 528.781,A -85,B 0,C 180,E1 -14935.064,E2 -14935.064} C_VEL
LIN {X 0,Y 327.041,Z 528.743,A -85,B 0,C 180,E1 -14937.536,E2 -14937.536} C_VEL
LIN {X 0,Y 327.21,Z 528.722,A -85,B 0,C 180,E1 -14939.999,E2 -14939.999} C_VEL
LIN {X 0,Y 327.062,Z 528.745,A -85,B 0,C 180,E1 -14942.463,E2 -14942.463} C_VEL
LIN {X 0,Y 326.957,Z 528.754,A -85,B 0,C 180,E1 -14946.586,E2 -14946.586} C_VEL
LIN {X 0,Y 326.798,Z 528.777,A -85,B 0,C 180,E1 -14949.906,E2 -14949.906} C_VEL
LIN {X 0,Y 326.751,Z 528.782,A -85,B 0,C 180,E1 -14953.685,E2 -14953.685} C_VEL
LIN {X 0,Y 326.691,Z 528.791,A -85,B 0,C 180,E1 -14957.528,E2 -14957.528} C_VEL
LIN {X 0,Y 326.657,Z 528.796,A -85,B 0,C 180,E1 -14960.135,E2 -14960.135} C_VEL
LIN {X 0,Y 326.657,Z 528.802,A -85,B 0,C 180,E1 -14964.128,E2 -14964.128} C_VEL
LIN {X 0,Y 326.699,Z 528.976,A -85,B 0,C 180,E1 -14965.321,E2 -14965.321} C_VEL
LIN {X 0,Y 327.316,Z 531.609,A -85,B 0,C 180,E1 -14966.328,E2 -14966.328} C_VEL
LIN {X 0,Y 335.364,Z 548.995,A -85,B 0,C 180,E1 -14967.588,E2 -14967.588} C_VEL
LIN {X 0,Y 339.443,Z 558.977,A -85,B 0,C 180,E1 -14968.219,E2 -14968.219} C_VEL
LIN {X 0,Y 337.209,Z 637.867,A -85,B 0,C 180,E1 -14970.07,E2 -14970.07} C_VEL
LIN {X 0,Y 336.449,Z 651.876,A -85,B 0,C 180,E1 -14970.661,E2 -14970.661} C_VEL
LIN {X 0,Y 335.592,Z 664.67,A -85,B 0,C 180,E1 -14971.477,E2 -14971.477} C_VEL
LIN {X 0,Y 334.385,Z 676.602,A -85,B 0,C 180,E1 -14972.493,E2 -14972.493} C_VEL
LIN {X 0,Y 333.19,Z 686.954,A -85,B 0,C 180,E1 -14973.62,E2 -14973.62} C_VEL
LIN {X 0,Y 331.911,Z 696.284,A -85,B 0,C 180,E1 -14974.869,E2 -14974.869} C_VEL
LIN {X 0,Y 330.488,Z 705.654,A -85,B 0,C 180,E1 -14976.414,E2 -14976.414} C_VEL
LIN {X 0,Y 329.095,Z 714.595,A -85,B 0,C 180,E1 -14978.265,E2 -14978.265} C_VEL
LIN {X 0,Y 327.975,Z 721.347,A -85,B 0,C 180,E1 -14980.004,E2 -14980.004} C_VEL
LIN {X 0,Y 327.049,Z 726.862,A -85,B 0,C 180,E1 -14981.771,E2 -14981.771} C_VEL
LIN {X 0,Y 326.34,Z 731.288,A -85,B 0,C 180,E1 -14983.562,E2 -14983.562} C_VEL
LIN {X 0,Y 325.814,Z 734.729,A -85,B 0,C 180,E1 -14985.383,E2 -14985.383} C_VEL
LIN {X 0,Y 325.356,Z 737.267,A -85,B 0,C 180,E1 -14987.258,E2 -14987.258} C_VEL
LIN {X 0,Y 325.027,Z 739.092,A -85,B 0,C 180,E1 -14989.559,E2 -14989.559} C_VEL
LIN {X 0,Y 324.882,Z 739.503,A -85,B 0,C 180,E1 -14991.147,E2 -14991.147} C_VEL
LIN {X 0,Y 324.86,Z 739.105,A -85,B 0,C 180,E1 -14993.172,E2 -14993.172} C_VEL
LIN {X 0,Y 324.999,Z 737.577,A -85,B 0,C 180,E1 -14995.258,E2 -14995.258} C_VEL
LIN {X 0,Y 325.37,Z 734.799,A -85,B 0,C 180,E1 -14997.393,E2 -14997.393} C_VEL
LIN {X 0,Y 325.885,Z 730.465,A -85,B 0,C 180,E1 -14999.612,E2 -14999.612} C_VEL
LIN {X 0,Y 326.545,Z 724.821,A -85,B 0,C 180,E1 -15001.74,E2 -15001.74} C_VEL
LIN {X 0,Y 327.397,Z 717.807,A -85,B 0,C 180,E1 -15003.777,E2 -15003.777} C_VEL
LIN {X 0,Y 328.413,Z 709.484,A -85,B 0,C 180,E1 -15005.673,E2 -15005.673} C_VEL
LIN {X 0,Y 329.439,Z 701.356,A -85,B 0,C 180,E1 -15007.175,E2 -15007.175} C_VEL
LIN {X 0,Y 330.552,Z 691.643,A -85,B 0,C 180,E1 -15008.648,E2 -15008.648} C_VEL
LIN {X 0,Y 331.771,Z 680.106,A -85,B 0,C 180,E1 -15010.034,E2 -15010.034} C_VEL
LIN {X 0,Y 332.748,Z 669.419,A -85,B 0,C 180,E1 -15011.051,E2 -15011.051} C_VEL
LIN {X 0,Y 333.635,Z 656.855,A -85,B 0,C 180,E1 -15011.978,E2 -15011.978} C_VEL
LIN {X 0,Y 334.325,Z 643.994,A -85,B 0,C 180,E1 -15012.648,E2 -15012.648} C_VEL
LIN {X 0,Y 334.755,Z 630.341,A -85,B 0,C 180,E1 -15013.104,E2 -15013.104} C_VEL
LIN {X 0,Y 336.411,Z 555.73,A -85,B 0,C 180,E1 -15014.793,E2 -15014.793} C_VEL
LIN {X 0,Y 327.44,Z 530.958,A -85,B 0,C 180,E1 -15015.998,E2 -15015.998} C_VEL
LIN {X 0,Y 326.838,Z 529.092,A -85,B 0,C 180,E1 -15016.105,E2 -15016.105} C_VEL
LIN {X 0,Y 326.779,Z 528.78,A -85,B 0,C 180,E1 -15016.316,E2 -15016.316} C_VEL
LIN {X 0,Y 326.809,Z 528.774,A -85,B 0,C 180,E1 -15020.094,E2 -15020.094} C_VEL
LIN {X 0,Y 326.963,Z 528.757,A -85,B 0,C 180,E1 -15022.59,E2 -15022.59} C_VEL
LIN {X 0,Y 326.774,Z 528.782,A -85,B 0,C 180,E1 -15025.065,E2 -15025.065} C_VEL
LIN {X 0,Y 327.045,Z 528.744,A -85,B 0,C 180,E1 -15027.537,E2 -15027.537} C_VEL
LIN {X 0,Y 327.196,Z 528.725,A -85,B 0,C 180,E1 -15030,E2 -15030} C_VEL
LIN {X 0,Y 327.045,Z 528.745,A -85,B 0,C 180,E1 -15032.463,E2 -15032.463} C_VEL
LIN {X 0,Y 326.994,Z 528.75,A -85,B 0,C 180,E1 -15036.169,E2 -15036.169} C_VEL
LIN {X 0,Y 326.911,Z 528.763,A -85,B 0,C 180,E1 -15038.655,E2 -15038.655} C_VEL
LIN {X 0,Y 326.731,Z 528.784,A -85,B 0,C 180,E1 -15042.421,E2 -15042.421} C_VEL
LIN {X 0,Y 326.751,Z 528.786,A -85,B 0,C 180,E1 -15044.957,E2 -15044.957} C_VEL
LIN {X 0,Y 326.729,Z 528.787,A -85,B 0,C 180,E1 -15048.838,E2 -15048.838} C_VEL
LIN {X 0,Y 326.616,Z 528.801,A -85,B 0,C 180,E1 -15052.787,E2 -15052.787} C_VEL
LIN {X 0,Y 326.686,Z 528.79,A -85,B 0,C 180,E1 -15055.483,E2 -15055.483} C_VEL
LIN {X 0,Y 326.657,Z 528.792,A -85,B 0,C 180,E1 -15059.659,E2 -15059.659} C_VEL
LIN {X 0,Y 326.618,Z 528.802,A -85,B 0,C 180,E1 -15062.947,E2 -15062.947} C_VEL
LIN {X 0,Y 326.589,Z 528.8,A -85,B 0,C 180,E1 -15066.306,E2 -15066.306} C_VEL
LIN {X 0,Y 325.948,Z 528.885,A -85,B 0,C 180,E1 -15067.336,E2 -15067.336} C_VEL
LIN {X 0,Y 323.132,Z 529.237,A -85,B 0,C 180,E1 -15069.012,E2 -15069.012} C_VEL
LIN {X 0,Y 320.726,Z 529.535,A -85,B 0,C 180,E1 -15070.371,E2 -15070.371} C_VEL
LIN {X 0,Y 319.68,Z 529.664,A -85,B 0,C 180,E1 -15071.422,E2 -15071.422} C_VEL
LIN {X 0,Y 319.589,Z 529.673,A -85,B 0,C 180,E1 -15071.778,E2 -15071.778} C_VEL
LIN {X 0,Y 319.639,Z 529.669,A -85,B 0,C 180,E1 -15075.285,E2 -15075.285} C_VEL
LIN {X 0,Y 319.576,Z 529.675,A -85,B 0,C 180,E1 -15078.72,E2 -15078.72} C_VEL
LIN {X 0,Y 319.576,Z 529.674,A -85,B 0,C 180,E1 -15082.343,E2 -15082.343} C_VEL
LIN {X 0,Y 319.553,Z 529.682,A -85,B 0,C 180,E1 -15085.123,E2 -15085.123} C_VEL
LIN {X 0,Y 319.563,Z 529.679,A -85,B 0,C 180,E1 -15089.058,E2 -15089.058} C_VEL
LIN {X 0,Y 319.601,Z 529.672,A -85,B 0,C 180,E1 -15092.498,E2 -15092.498} C_VEL
LIN {X 0,Y 319.596,Z 529.675,A -85,B 0,C 180,E1 -15095.304,E2 -15095.304} C_VEL
LIN {X 0,Y 319.594,Z 529.673,A -85,B 0,C 180,E1 -15099.4,E2 -15099.4} C_VEL
LIN {X 0,Y 319.65,Z 529.664,A -85,B 0,C 180,E1 -15102.073,E2 -15102.073} C_VEL
LIN {X 0,Y 319.725,Z 529.655,A -85,B 0,C 180,E1 -15106.008,E2 -15106.008} C_VEL
LIN {X 0,Y 319.752,Z 529.65,A -85,B 0,C 180,E1 -15109.873,E2 -15109.873} C_VEL
LIN {X 0,Y 319.927,Z 529.629,A -85,B 0,C 180,E1 -15112.427,E2 -15112.427} C_VEL
LIN {X 0,Y 319.745,Z 529.656,A -85,B 0,C 180,E1 -15114.957,E2 -15114.957} C_VEL
LIN {X 0,Y 319.985,Z 529.625,A -85,B 0,C 180,E1 -15117.483,E2 -15117.483} C_VEL
LIN {X 0,Y 320.162,Z 529.599,A -85,B 0,C 180,E1 -15120.001,E2 -15120.001} C_VEL
LIN {X 0,Y 320.011,Z 529.619,A -85,B 0,C 180,E1 -15122.518,E2 -15122.518} C_VEL
LIN {X 0,Y 319.94,Z 529.628,A -85,B 0,C 180,E1 -15126.306,E2 -15126.306} C_VEL
LIN {X 0,Y 319.831,Z 529.644,A -85,B 0,C 180,E1 -15128.849,E2 -15128.849} C_VEL
LIN {X 0,Y 319.675,Z 529.663,A -85,B 0,C 180,E1 -15132.701,E2 -15132.701} C_VEL
LIN {X 0,Y 319.693,Z 529.664,A -85,B 0,C 180,E1 -15135.296,E2 -15135.296} C_VEL
LIN {X 0,Y 319.669,Z 529.668,A -85,B 0,C 180,E1 -15139.256,E2 -15139.256} C_VEL
LIN {X 0,Y 319.565,Z 529.68,A -85,B 0,C 180,E1 -15143.32,E2 -15143.32} C_VEL
LIN {X 0,Y 319.63,Z 529.667,A -85,B 0,C 180,E1 -15146.089,E2 -15146.089} C_VEL
LIN {X 0,Y 319.586,Z 529.675,A -85,B 0,C 180,E1 -15148.935,E2 -15148.935} C_VEL
LIN {X 0,Y 319.535,Z 529.68,A -85,B 0,C 180,E1 -15151.862,E2 -15151.862} C_VEL
LIN {X 0,Y 319.577,Z 529.678,A -85,B 0,C 180,E1 -15155.544,E2 -15155.544} C_VEL
LIN {X 0,Y 319.555,Z 529.677,A -85,B 0,C 180,E1 -15158.011,E2 -15158.011} C_VEL
LIN {X 0,Y 319.524,Z 529.684,A -85,B 0,C 180,E1 -15161.598,E2 -15161.598} C_VEL
LIN {X 0,Y 319.569,Z 529.68,A -85,B 0,C 180,E1 -15165.273,E2 -15165.273} C_VEL
LIN {X 0,Y 319.578,Z 529.675,A -85,B 0,C 180,E1 -15168.721,E2 -15168.721} C_VEL
LIN {X 0,Y 319.598,Z 529.672,A -85,B 0,C 180,E1 -15172.34,E2 -15172.34} C_VEL
LIN {X 0,Y 319.576,Z 529.679,A -85,B 0,C 180,E1 -15176.46,E2 -15176.46} C_VEL
LIN {X 0,Y 319.633,Z 530.044,A -85,B 0,C 180,E1 -15176.672,E2 -15176.672} C_VEL
LIN {X 0,Y 322.147,Z 541.357,A -85,B 0,C 180,E1 -15179.884,E2 -15179.884} C_VEL
LIN {X 0,Y 324.377,Z 552.641,A -85,B 0,C 180,E1 -15182.937,E2 -15182.937} C_VEL
LIN {X 0,Y 323.599,Z 560.813,A -85,B 0,C 180,E1 -15184.945,E2 -15184.945} C_VEL
LIN {X 0,Y 323.197,Z 563.761,A -85,B 0,C 180,E1 -15185.656,E2 -15185.656} C_VEL
LIN {X 0,Y 329.028,Z 606.364,A -85,B 0,C 180,E1 -15187.107,E2 -15187.107} C_VEL
LIN {X 0,Y 327.478,Z 673.189,A -85,B 0,C 180,E1 -15188.686,E2 -15188.686} C_VEL
LIN {X 0,Y 326.642,Z 686.72,A -85,B 0,C 180,E1 -15189.248,E2 -15189.248} C_VEL
LIN {X 0,Y 325.528,Z 699.571,A -85,B 0,C 180,E1 -15190.039,E2 -15190.039} C_VEL
LIN {X 0,Y 324.379,Z 711.356,A -85,B 0,C 180,E1 -15191.036,E2 -15191.036} C_VEL
LIN {X 0,Y 323.074,Z 722.749,A -85,B 0,C 180,E1 -15192.269,E2 -15192.269} C_VEL
LIN {X 0,Y 321.849,Z 733.051,A -85,B 0,C 180,E1 -15193.674,E2 -15193.674} C_VEL
LIN {X 0,Y 320.89,Z 741.475,A -85,B 0,C 180,E1 -15195.088,E2 -15195.088} C_VEL
LIN {X 0,Y 319.722,Z 750.621,A -85,B 0,C 180,E1 -15196.979,E2 -15196.979} C_VEL
LIN {X 0,Y 318.811,Z 757.982,A -85,B 0,C 180,E1 -15198.879,E2 -15198.879} C_VEL
LIN {X 0,Y 318.39,Z 762.957,A -85,B 0,C 180,E1 -15200.471,E2 -15200.471} C_VEL
LIN {X 0,Y 318.081,Z 767.774,A -85,B 0,C 180,E1 -15202.382,E2 -15202.382} C_VEL
LIN {X 0,Y 317.944,Z 771.12,A -85,B 0,C 180,E1 -15204.105,E2 -15204.105} C_VEL
LIN {X 0,Y 317.923,Z 774.049,A -85,B 0,C 180,E1 -15206.198,E2 -15206.198} C_VEL
LIN {X 0,Y 317.92,Z 775.261,A -85,B 0,C 180,E1 -15207.466,E2 -15207.466} C_VEL
LIN {X 0,Y 318.021,Z 776.027,A -85,B 0,C 180,E1 -15208.734,E2 -15208.734} C_VEL
LIN {X 0,Y 318.112,Z 776.369,A -85,B 0,C 180,E1 -15210,E2 -15210} C_VEL
LIN {X 0,Y 318.011,Z 776.299,A -85,B 0,C 180,E1 -15211.266,E2 -15211.266} C_VEL
LIN {X 0,Y 317.897,Z 775.831,A -85,B 0,C 180,E1 -15212.534,E2 -15212.534} C_VEL
LIN {X 0,Y 317.905,Z 774.93,A -85,B 0,C 180,E1 -15213.803,E2 -15213.803} C_VEL
LIN {X 0,Y 317.876,Z 772.707,A -85,B 0,C 180,E1 -15215.776,E2 -15215.776} C_VEL
LIN {X 0,Y 318.036,Z 769.69,A -85,B 0,C 180,E1 -15217.619,E2 -15217.619} C_VEL
LIN {X 0,Y 318.413,Z 765.518,A -85,B 0,C 180,E1 -15219.528,E2 -15219.528} C_VEL
LIN {X 0,Y 319.158,Z 759.154,A -85,B 0,C 180,E1 -15221.752,E2 -15221.752} C_VEL
LIN {X 0,Y 320.242,Z 752.265,A -85,B 0,C 180,E1 -15223.645,E2 -15223.645} C_VEL
LIN {X 0,Y 321.3,Z 745.271,A -85,B 0,C 180,E1 -15225.217,E2 -15225.217} C_VEL
LIN {X 0,Y 322.54,Z 736.878,A -85,B 0,C 180,E1 -15226.78,E2 -15226.78} C_VEL
LIN {X 0,Y 324.09,Z 726.65,A -85,B 0,C 180,E1 -15228.326,E2 -15228.326} C_VEL
LIN {X 0,Y 325.747,Z 715.124,A -85,B 0,C 180,E1 -15229.7,E2 -15229.7} C_VEL
LIN {X 0,Y 327.226,Z 703.866,A -85,B 0,C 180,E1 -15230.755,E2 -15230.755} C_VEL
LIN {X 0,Y 328.561,Z 691.288,A -85,B 0,C 180,E1 -15231.652,E2 -15231.652} C_VEL
LIN {X 0,Y 329.762,Z 678.03,A -85,B 0,C 180,E1 -15232.31,E2 -15232.31} C_VEL
LIN {X 0,Y 330.473,Z 665.2,A -85,B 0,C 180,E1 -15232.718,E2 -15232.718} C_VEL
LIN {X 0,Y 331.933,Z 606.783,A -85,B 0,C 180,E1 -15234.107,E2 -15234.107} C_VEL
LIN {X 0,Y 328.904,Z 583.706,A -85,B 0,C 180,E1 -15234.995,E2 -15234.995} C_VEL
LIN {X 0,Y 325.176,Z 563.928,A -85,B 0,C 180,E1 -15235.89,E2 -15235.89} C_VEL
LIN {X 0,Y 324.668,Z 561.502,A -85,B 0,C 180,E1 -15236.009,E2 -15236.009} C_VEL
LIN {X 0,Y 325.373,Z 555.947,A -85,B 0,C 180,E1 -15237.418,E2 -15237.418} C_VEL
LIN {X 0,Y 323.742,Z 547.199,A -85,B 0,C 180,E1 -15239.953,E2 -15239.953} C_VEL
LIN {X 0,Y 321.423,Z 536.913,A -85,B 0,C 180,E1 -15243.135,E2 -15243.135} C_VEL
LIN {X 0,Y 319.577,Z 529.681,A -85,B 0,C 180,E1 -15245.609,E2 -15245.609} C_VEL
LIN {X 0,Y 319.599,Z 529.676,A -85,B 0,C 180,E1 -15248.003,E2 -15248.003} C_VEL
LIN {X 0,Y 319.596,Z 529.675,A -85,B 0,C 180,E1 -15251.61,E2 -15251.61} C_VEL
LIN {X 0,Y 319.542,Z 529.679,A -85,B 0,C 180,E1 -15255.266,E2 -15255.266} C_VEL
LIN {X 0,Y 319.527,Z 529.684,A -85,B 0,C 180,E1 -15258.711,E2 -15258.711} C_VEL
LIN {X 0,Y 319.575,Z 529.676,A -85,B 0,C 180,E1 -15262.343,E2 -15262.343} C_VEL
LIN {X 0,Y 319.557,Z 529.677,A -85,B 0,C 180,E1 -15265.122,E2 -15265.122} C_VEL
LIN {X 0,Y 319.566,Z 529.674,A -85,B 0,C 180,E1 -15269.057,E2 -15269.057} C_VEL
LIN {X 0,Y 319.604,Z 529.668,A -85,B 0,C 180,E1 -15272.497,E2 -15272.497} C_VEL
LIN {X 0,Y 319.599,Z 529.667,A -85,B 0,C 180,E1 -15275.303,E2 -15275.303} C_VEL
LIN {X 0,Y 319.591,Z 529.674,A -85,B 0,C 180,E1 -15278.047,E2 -15278.047} C_VEL
LIN {X 0,Y 319.683,Z 529.666,A -85,B 0,C 180,E1 -15280.961,E2 -15280.961} C_VEL
LIN {X 0,Y 319.725,Z 529.657,A -85,B 0,C 180,E1 -15285.275,E2 -15285.275} C_VEL
LIN {X 0,Y 319.75,Z 529.649,A -85,B 0,C 180,E1 -15289.872,E2 -15289.872} C_VEL
LIN {X 0,Y 319.92,Z 529.634,A -85,B 0,C 180,E1 -15292.425,E2 -15292.425} C_VEL
LIN {X 0,Y 319.744,Z 529.655,A -85,B 0,C 180,E1 -15294.955,E2 -15294.955} C_VEL
LIN {X 0,Y 319.985,Z 529.622,A -85,B 0,C 180,E1 -15297.482,E2 -15297.482} C_VEL
LIN {X 0,Y 320.162,Z 529.6,A -85,B 0,C 180,E1 -15299.999,E2 -15299.999} C_VEL
LIN {X 0,Y 320.002,Z 529.625,A -85,B 0,C 180,E1 -15302.517,E2 -15302.517} C_VEL
LIN {X 0,Y 319.92,Z 529.63,A -85,B 0,C 180,E1 -15306.572,E2 -15306.572} C_VEL
LIN {X 0,Y 319.745,Z 529.656,A -85,B 0,C 180,E1 -15310.127,E2 -15310.127} C_VEL
LIN {X 0,Y 319.723,Z 529.661,A -85,B 0,C 180,E1 -15314.724,E2 -15314.724} C_VEL
LIN {X 0,Y 319.681,Z 529.665,A -85,B 0,C 180,E1 -15319.037,E2 -15319.037} C_VEL
LIN {X 0,Y 319.567,Z 529.684,A -85,B 0,C 180,E1 -15323.319,E2 -15323.319} C_VEL
LIN {X 0,Y 319.673,Z 529.854,A -85,B 0,C 180,E1 -15324.69,E2 -15324.69} C_VEL
LIN {X 0,Y 320.192,Z 532.142,A -85,B 0,C 180,E1 -15325.601,E2 -15325.601} C_VEL
LIN {X 0,Y 328.802,Z 550.222,A -85,B 0,C 180,E1 -15326.997,E2 -15326.997} C_VEL
LIN {X 0,Y 333.157,Z 560.906,A -85,B 0,C 180,E1 -15327.696,E2 -15327.696} C_VEL
LIN {X 0,Y 330.805,Z 638.471,A -85,B 0,C 180,E1 -15329.556,E2 -15329.556} C_VEL
LIN {X 0,Y 330.041,Z 652.048,A -85,B 0,C 180,E1 -15330.141,E2 -15330.141} C_VEL
LIN {X 0,Y 329.126,Z 664.714,A -85,B 0,C 180,E1 -15330.955,E2 -15330.955} C_VEL
LIN {X 0,Y 327.928,Z 676.271,A -85,B 0,C 180,E1 -15331.949,E2 -15331.949} C_VEL
LIN {X 0,Y 326.576,Z 687.466,A -85,B 0,C 180,E1 -15333.18,E2 -15333.18} C_VEL
LIN {X 0,Y 325.241,Z 696.705,A -85,B 0,C 180,E1 -15334.44,E2 -15334.44} C_VEL
LIN {X 0,Y 323.915,Z 705.246,A -85,B 0,C 180,E1 -15335.86,E2 -15335.86} C_VEL
LIN {X 0,Y 322.485,Z 713.749,A -85,B 0,C 180,E1 -15337.604,E2 -15337.604} C_VEL
LIN {X 0,Y 321.119,Z 721.751,A -85,B 0,C 180,E1 -15339.671,E2 -15339.671} C_VEL
LIN {X 0,Y 320.025,Z 727.89,A -85,B 0,C 180,E1 -15341.699,E2 -15341.699} C_VEL
LIN {X 0,Y 319.315,Z 731.96,A -85,B 0,C 180,E1 -15343.423,E2 -15343.423} C_VEL
LIN {X 0,Y 318.805,Z 735.091,A -85,B 0,C 180,E1 -15345.137,E2 -15345.137} C_VEL
LIN {X 0,Y 318.387,Z 737.385,A -85,B 0,C 180,E1 -15346.822,E2 -15346.822} C_VEL
LIN {X 0,Y 318.036,Z 739.076,A -85,B 0,C 180,E1 -15348.705,E2 -15348.705} C_VEL
LIN {X 0,Y 317.814,Z 739.887,A -85,B 0,C 180,E1 -15350.711,E2 -15350.711} C_VEL
LIN {X 0,Y 317.76,Z 739.672,A -85,B 0,C 180,E1 -15352.77,E2 -15352.77} C_VEL
LIN {X 0,Y 317.885,Z 738.317,A -85,B 0,C 180,E1 -15354.914,E2 -15354.914} C_VEL
LIN {X 0,Y 318.198,Z 735.772,A -85,B 0,C 180,E1 -15357.065,E2 -15357.065} C_VEL
LIN {X 0,Y 318.784,Z 731.297,A -85,B 0,C 180,E1 -15359.532,E2 -15359.532} C_VEL
LIN {X 0,Y 319.416,Z 725.918,A -85,B 0,C 180,E1 -15361.654,E2 -15361.654} C_VEL
LIN {X 0,Y 320.215,Z 719.536,A -85,B 0,C 180,E1 -15363.613,E2 -15363.613} C_VEL
LIN {X 0,Y 321.2,Z 712.118,A -85,B 0,C 180,E1 -15365.435,E2 -15365.435} C_VEL
LIN {X 0,Y 322.389,Z 702.935,A -85,B 0,C 180,E1 -15367.236,E2 -15367.236} C_VEL
LIN {X 0,Y 323.523,Z 693.645,A -85,B 0,C 180,E1 -15368.712,E2 -15368.712} C_VEL
LIN {X 0,Y 324.65,Z 683.158,A -85,B 0,C 180,E1 -15370.065,E2 -15370.065} C_VEL
LIN {X 0,Y 325.794,Z 671.516,A -85,B 0,C 180,E1 -15371.248,E2 -15371.248} C_VEL
LIN {X 0,Y 326.769,Z 658.368,A -85,B 0,C 180,E1 -15372.267,E2 -15372.267} C_VEL
LIN {X 0,Y 327.492,Z 645.966,A -85,B 0,C 180,E1 -15372.959,E2 -15372.959} C_VEL
LIN {X 0,Y 327.963,Z 633.171,A -85,B 0,C 180,E1 -15373.425,E2 -15373.425} C_VEL
LIN {X 0,Y 329.801,Z 557.224,A -85,B 0,C 180,E1 -15375.184,E2 -15375.184} C_VEL
LIN {X 0,Y 320.813,Z 532.696,A -85,B 0,C 180,E1 -15376.42,E2 -15376.42} C_VEL
LIN {X 0,Y 319.72,Z 529.696,A -85,B 0,C 180,E1 -15376.575,E2 -15376.575} C_VEL
LIN {X 0,Y 319.754,Z 529.654,A -85,B 0,C 180,E1 -15379.873,E2 -15379.873} C_VEL
LIN {X 0,Y 319.922,Z 529.634,A -85,B 0,C 180,E1 -15382.426,E2 -15382.426} C_VEL
LIN {X 0,Y 319.744,Z 529.659,A -85,B 0,C 180,E1 -15384.956,E2 -15384.956} C_VEL
LIN {X 0,Y 319.989,Z 529.624,A -85,B 0,C 180,E1 -15387.482,E2 -15387.482} C_VEL
LIN {X 0,Y 320.148,Z 529.603,A -85,B 0,C 180,E1 -15390,E2 -15390} C_VEL
LIN {X 0,Y 319.989,Z 529.625,A -85,B 0,C 180,E1 -15392.518,E2 -15392.518} C_VEL
LIN {X 0,Y 319.949,Z 529.628,A -85,B 0,C 180,E1 -15396.305,E2 -15396.305} C_VEL
LIN {X 0,Y 319.84,Z 529.646,A -85,B 0,C 180,E1 -15398.848,E2 -15398.848} C_VEL
LIN {X 0,Y 319.679,Z 529.664,A -85,B 0,C 180,E1 -15402.7,E2 -15402.7} C_VEL
LIN {X 0,Y 319.696,Z 529.661,A -85,B 0,C 180,E1 -15405.295,E2 -15405.295} C_VEL
LIN {X 0,Y 319.671,Z 529.665,A -85,B 0,C 180,E1 -15409.255,E2 -15409.255} C_VEL
LIN {X 0,Y 319.566,Z 529.678,A -85,B 0,C 180,E1 -15413.319,E2 -15413.319} C_VEL
LIN {X 0,Y 319.631,Z 529.667,A -85,B 0,C 180,E1 -15416.088,E2 -15416.088} C_VEL
LIN {X 0,Y 319.586,Z 529.678,A -85,B 0,C 180,E1 -15418.933,E2 -15418.933} C_VEL
LIN {X 0,Y 319.534,Z 529.679,A -85,B 0,C 180,E1 -15421.861,E2 -15421.861} C_VEL
LIN {X 0,Y 319.575,Z 529.675,A -85,B 0,C 180,E1 -15425.543,E2 -15425.543} C_VEL
LIN {X 0,Y 319.595,Z 529.671,A -85,B 0,C 180,E1 -15428.004,E2 -15428.004} C_VEL
LIN {X 0,Y 319.589,Z 529.673,A -85,B 0,C 180,E1 -15431.778,E2 -15431.778} C_VEL
LIN {X 0,Y 318.899,Z 529.762,A -85,B 0,C 180,E1 -15432.829,E2 -15432.829} C_VEL
LIN {X 0,Y 316.029,Z 530.117,A -85,B 0,C 180,E1 -15434.54,E2 -15434.54} C_VEL
LIN {X 0,Y 313.623,Z 530.415,A -85,B 0,C 180,E1 -15435.927,E2 -15435.927} C_VEL
LIN {X 0,Y 312.614,Z 530.545,A -85,B 0,C 180,E1 -15437.001,E2 -15437.001} C_VEL
LIN {X 0,Y 312.544,Z 530.547,A -85,B 0,C 180,E1 -15437.364,E2 -15437.364} C_VEL
LIN {X 0,Y 312.526,Z 530.556,A -85,B 0,C 180,E1 -15440.976,E2 -15440.976} C_VEL
LIN {X 0,Y 312.525,Z 530.552,A -85,B 0,C 180,E1 -15444.22,E2 -15444.22} C_VEL
LIN {X 0,Y 312.497,Z 530.556,A -85,B 0,C 180,E1 -15447.334,E2 -15447.334} C_VEL
LIN {X 0,Y 312.545,Z 530.554,A -85,B 0,C 180,E1 -15451.276,E2 -15451.276} C_VEL
LIN {X 0,Y 312.577,Z 530.548,A -85,B 0,C 180,E1 -15454.711,E2 -15454.711} C_VEL
LIN {X 0,Y 312.529,Z 530.553,A -85,B 0,C 180,E1 -15458.913,E2 -15458.913} C_VEL
LIN {X 0,Y 312.63,Z 530.54,A -85,B 0,C 180,E1 -15461.657,E2 -15461.657} C_VEL
LIN {X 0,Y 312.686,Z 530.533,A -85,B 0,C 180,E1 -15465.687,E2 -15465.687} C_VEL
LIN {X 0,Y 312.696,Z 530.529,A -85,B 0,C 180,E1 -15469.642,E2 -15469.642} C_VEL
LIN {X 0,Y 312.865,Z 530.508,A -85,B 0,C 180,E1 -15472.255,E2 -15472.255} C_VEL
LIN {X 0,Y 312.715,Z 530.53,A -85,B 0,C 180,E1 -15474.843,E2 -15474.843} C_VEL
LIN {X 0,Y 312.985,Z 530.495,A -85,B 0,C 180,E1 -15478.714,E2 -15478.714} C_VEL
LIN {X 0,Y 313.113,Z 530.477,A -85,B 0,C 180,E1 -15480.001,E2 -15480.001} C_VEL
LIN {X 0,Y 312.955,Z 530.498,A -85,B 0,C 180,E1 -15482.575,E2 -15482.575} C_VEL
LIN {X 0,Y 312.897,Z 530.506,A -85,B 0,C 180,E1 -15486.449,E2 -15486.449} C_VEL
LIN {X 0,Y 312.761,Z 530.526,A -85,B 0,C 180,E1 -15489.051,E2 -15489.051} C_VEL
LIN {X 0,Y 312.628,Z 530.542,A -85,B 0,C 180,E1 -15492.992,E2 -15492.992} C_VEL
LIN {X 0,Y 312.632,Z 530.54,A -85,B 0,C 180,E1 -15495.651,E2 -15495.651} C_VEL
LIN {X 0,Y 312.625,Z 530.545,A -85,B 0,C 180,E1 -15499.237,E2 -15499.237} C_VEL
LIN {X 0,Y 312.541,Z 530.552,A -85,B 0,C 180,E1 -15502.79,E2 -15502.79} C_VEL
LIN {X 0,Y 312.598,Z 530.544,A -85,B 0,C 180,E1 -15505.937,E2 -15505.937} C_VEL
LIN {X 0,Y 312.543,Z 530.552,A -85,B 0,C 180,E1 -15509.651,E2 -15509.651} C_VEL
LIN {X 0,Y 312.517,Z 530.555,A -85,B 0,C 180,E1 -15513.69,E2 -15513.69} C_VEL
LIN {X 0,Y 312.535,Z 530.556,A -85,B 0,C 180,E1 -15517.384,E2 -15517.384} C_VEL
LIN {X 0,Y 312.488,Z 530.558,A -85,B 0,C 180,E1 -15520.71,E2 -15520.71} C_VEL
LIN {X 0,Y 312.517,Z 530.554,A -85,B 0,C 180,E1 -15524.199,E2 -15524.199} C_VEL
LIN {X 0,Y 312.547,Z 530.551,A -85,B 0,C 180,E1 -15527.907,E2 -15527.907} C_VEL
LIN {X 0,Y 312.558,Z 530.55,A -85,B 0,C 180,E1 -15531.906,E2 -15531.906} C_VEL
LIN {X 0,Y 312.547,Z 530.553,A -85,B 0,C 180,E1 -15536.15,E2 -15536.15} C_VEL
LIN {X 0,Y 315.259,Z 543.035,A -85,B 0,C 180,E1 -15539.798,E2 -15539.798} C_VEL
LIN {X 0,Y 317.337,Z 553.167,A -85,B 0,C 180,E1 -15542.608,E2 -15542.608} C_VEL
LIN {X 0,Y 317.321,Z 556.057,A -85,B 0,C 180,E1 -15543.353,E2 -15543.353} C_VEL
LIN {X 0,Y 316.373,Z 563.458,A -85,B 0,C 180,E1 -15545.18,E2 -15545.18} C_VEL
LIN {X 0,Y 322.287,Z 606.652,A -85,B 0,C 180,E1 -15546.686,E2 -15546.686} C_VEL
LIN {X 0,Y 320.741,Z 673.148,A -85,B 0,C 180,E1 -15548.3,E2 -15548.3} C_VEL
LIN {X 0,Y 319.891,Z 686.56,A -85,B 0,C 180,E1 -15548.873,E2 -15548.873} C_VEL
LIN {X 0,Y 318.739,Z 699.328,A -85,B 0,C 180,E1 -15549.68,E2 -15549.68} C_VEL
LIN {X 0,Y 317.451,Z 711.872,A -85,B 0,C 180,E1 -15550.773,E2 -15550.773} C_VEL
LIN {X 0,Y 316.113,Z 723.1,A -85,B 0,C 180,E1 -15552.033,E2 -15552.033} C_VEL
LIN {X 0,Y 314.884,Z 732.997,A -85,B 0,C 180,E1 -15553.431,E2 -15553.431} C_VEL
LIN {X 0,Y 313.771,Z 742.38,A -85,B 0,C 180,E1 -15555.074,E2 -15555.074} C_VEL
LIN {X 0,Y 312.582,Z 751.309,A -85,B 0,C 180,E1 -15557.007,E2 -15557.007} C_VEL
LIN {X 0,Y 311.701,Z 758.434,A -85,B 0,C 180,E1 -15558.951,E2 -15558.951} C_VEL
LIN {X 0,Y 311.218,Z 764.125,A -85,B 0,C 180,E1 -15560.905,E2 -15560.905} C_VEL
LIN {X 0,Y 310.933,Z 768.578,A -85,B 0,C 180,E1 -15562.859,E2 -15562.859} C_VEL
LIN {X 0,Y 310.821,Z 771.919,A -85,B 0,C 180,E1 -15564.811,E2 -15564.811} C_VEL
LIN {X 0,Y 310.85,Z 773.569,A -85,B 0,C 180,E1 -15566.111,E2 -15566.111} C_VEL
LIN {X 0,Y 310.834,Z 774.797,A -85,B 0,C 180,E1 -15567.408,E2 -15567.408} C_VEL
LIN {X 0,Y 310.926,Z 775.593,A -85,B 0,C 180,E1 -15568.705,E2 -15568.705} C_VEL
LIN {X 0,Y 311.023,Z 775.949,A -85,B 0,C 180,E1 -15570,E2 -15570} C_VEL
LIN {X 0,Y 310.916,Z 775.893,A -85,B 0,C 180,E1 -15571.295,E2 -15571.295} C_VEL
LIN {X 0,Y 310.812,Z 775.44,A -85,B 0,C 180,E1 -15572.592,E2 -15572.592} C_VEL
LIN {X 0,Y 310.808,Z 774.566,A -85,B 0,C 180,E1 -15573.89,E2 -15573.89} C_VEL
LIN {X 0,Y 310.794,Z 772.594,A -85,B 0,C 180,E1 -15575.742,E2 -15575.742} C_VEL
LIN {X 0,Y 310.983,Z 769.386,A -85,B 0,C 180,E1 -15577.793,E2 -15577.793} C_VEL
LIN {X 0,Y 311.365,Z 765.252,A -85,B 0,C 180,E1 -15579.746,E2 -15579.746} C_VEL
LIN {X 0,Y 312.175,Z 758.941,A -85,B 0,C 180,E1 -15582.019,E2 -15582.019} C_VEL
LIN {X 0,Y 313.326,Z 752.092,A -85,B 0,C 180,E1 -15583.953,E2 -15583.953} C_VEL
LIN {X 0,Y 314.669,Z 743.817,A -85,B 0,C 180,E1 -15585.837,E2 -15585.837} C_VEL
LIN {X 0,Y 316.048,Z 734.968,A -85,B 0,C 180,E1 -15587.469,E2 -15587.469} C_VEL
LIN {X 0,Y 317.7,Z 724.333,A -85,B 0,C 180,E1 -15589.043,E2 -15589.043} C_VEL
LIN {X 0,Y 319.512,Z 712.431,A -85,B 0,C 180,E1 -15590.437,E2 -15590.437} C_VEL
LIN {X 0,Y 321.08,Z 700.496,A -85,B 0,C 180,E1 -15591.508,E2 -15591.508} C_VEL
LIN {X 0,Y 322.403,Z 688.209,A -85,B 0,C 180,E1 -15592.34,E2 -15592.34} C_VEL
LIN {X 0,Y 323.513,Z 675.756,A -85,B 0,C 180,E1 -15592.934,E2 -15592.934} C_VEL
LIN {X 0,Y 324.181,Z 661.433,A -85,B 0,C 180,E1 -15593.356,E2 -15593.356} C_VEL
LIN {X 0,Y 325.585,Z 607.17,A -85,B 0,C 180,E1 -15594.674,E2 -15594.674} C_VEL
LIN {X 0,Y 322.541,Z 584.103,A -85,B 0,C 180,E1 -15595.594,E2 -15595.594} C_VEL
LIN {X 0,Y 319.068,Z 565.692,A -85,B 0,C 180,E1 -15596.467,E2 -15596.467} C_VEL
LIN {X 0,Y 318.163,Z 560.866,A -85,B 0,C 180,E1 -15596.74,E2 -15596.74} C_VEL
LIN {X 0,Y 318.561,Z 557.577,A -85,B 0,C 180,E1 -15597.599,E2 -15597.599} C_VEL
LIN {X 0,Y 316.942,Z 549.045,A -85,B 0,C 180,E1 -15600.139,E2 -15600.139} C_VEL
LIN {X 0,Y 314.501,Z 538.278,A -85,B 0,C 180,E1 -15603.577,E2 -15603.577} C_VEL
LIN {X 0,Y 312.525,Z 530.56,A -85,B 0,C 180,E1 -15606.313,E2 -15606.313} C_VEL
LIN {X 0,Y 312.538,Z 530.553,A -85,B 0,C 180,E1 -15609.022,E2 -15609.022} C_VEL
LIN {X 0,Y 312.548,Z 530.553,A -85,B 0,C 180,E1 -15612.421,E2 -15612.421} C_VEL
LIN {X 0,Y 312.512,Z 530.556,A -85,B 0,C 180,E1 -15616.023,E2 -15616.023} C_VEL
LIN {X 0,Y 312.502,Z 530.555,A -85,B 0,C 180,E1 -15619.873,E2 -15619.873} C_VEL
LIN {X 0,Y 312.535,Z 530.551,A -85,B 0,C 180,E1 -15622.615,E2 -15622.615} C_VEL
LIN {X 0,Y 312.516,Z 530.551,A -85,B 0,C 180,E1 -15626.31,E2 -15626.31} C_VEL
LIN {X 0,Y 312.541,Z 530.552,A -85,B 0,C 180,E1 -15630.349,E2 -15630.349} C_VEL
LIN {X 0,Y 312.598,Z 530.546,A -85,B 0,C 180,E1 -15634.063,E2 -15634.063} C_VEL
LIN {X 0,Y 312.582,Z 530.548,A -85,B 0,C 180,E1 -15637.528,E2 -15637.528} C_VEL
LIN {X 0,Y 312.632,Z 530.54,A -85,B 0,C 180,E1 -15641.655,E2 -15641.655} C_VEL
LIN {X 0,Y 312.688,Z 530.531,A -85,B 0,C 180,E1 -15645.685,E2 -15645.685} C_VEL
LIN {X 0,Y 312.695,Z 530.528,A -85,B 0,C 180,E1 -15649.641,E2 -15649.641} C_VEL
LIN {X 0,Y 312.861,Z 530.513,A -85,B 0,C 180,E1 -15652.253,E2 -15652.253} C_VEL
LIN {X 0,Y 312.714,Z 530.529,A -85,B 0,C 180,E1 -15654.842,E2 -15654.842} C_VEL
LIN {X 0,Y 312.985,Z 530.499,A -85,B 0,C 180,E1 -15658.713,E2 -15658.713} C_VEL
LIN {X 0,Y 313.114,Z 530.478,A -85,B 0,C 180,E1 -15659.999,E2 -15659.999} C_VEL
LIN {X 0,Y 312.946,Z 530.504,A -85,B 0,C 180,E1 -15662.574,E2 -15662.574} C_VEL
LIN {X 0,Y 312.886,Z 530.506,A -85,B 0,C 180,E1 -15666.551,E2 -15666.551} C_VEL
LIN {X 0,Y 312.76,Z 530.524,A -85,B 0,C 180,E1 -15669.049,E2 -15669.049} C_VEL
LIN {X 0,Y 312.627,Z 530.545,A -85,B 0,C 180,E1 -15672.991,E2 -15672.991} C_VEL
LIN {X 0,Y 312.63,Z 530.542,A -85,B 0,C 180,E1 -15675.649,E2 -15675.649} C_VEL
LIN {X 0,Y 312.623,Z 530.543,A -85,B 0,C 180,E1 -15679.236,E2 -15679.236} C_VEL
LIN {X 0,Y 312.576,Z 530.557,A -85,B 0,C 180,E1 -15683.872,E2 -15683.872} C_VEL
LIN {X 0,Y 313.176,Z 532.87,A -85,B 0,C 180,E1 -15684.838,E2 -15684.838} C_VEL
LIN {X 0,Y 321.154,Z 549.154,A -85,B 0,C 180,E1 -15686.188,E2 -15686.188} C_VEL
LIN {X 0,Y 326.854,Z 562.661,A -85,B 0,C 180,E1 -15687.144,E2 -15687.144} C_VEL
LIN {X 0,Y 324.461,Z 638.878,A -85,B 0,C 180,E1 -15689.011,E2 -15689.011} C_VEL
LIN {X 0,Y 323.647,Z 652.45,A -85,B 0,C 180,E1 -15689.604,E2 -15689.604} C_VEL
LIN {X 0,Y 322.699,Z 664.973,A -85,B 0,C 180,E1 -15690.421,E2 -15690.421} C_VEL
LIN {X 0,Y 321.404,Z 677.081,A -85,B 0,C 180,E1 -15691.485,E2 -15691.485} C_VEL
LIN {X 0,Y 319.997,Z 687.98,A -85,B 0,C 180,E1 -15692.713,E2 -15692.713} C_VEL
LIN {X 0,Y 318.553,Z 697.498,A -85,B 0,C 180,E1 -15694.043,E2 -15694.043} C_VEL
LIN {X 0,Y 317.076,Z 706.364,A -85,B 0,C 180,E1 -15695.57,E2 -15695.57} C_VEL
LIN {X 0,Y 315.649,Z 714.537,A -85,B 0,C 180,E1 -15697.307,E2 -15697.307} C_VEL
LIN {X 0,Y 314.385,Z 721.489,A -85,B 0,C 180,E1 -15699.129,E2 -15699.129} C_VEL
LIN {X 0,Y 313.325,Z 727.088,A -85,B 0,C 180,E1 -15700.951,E2 -15700.951} C_VEL
LIN {X 0,Y 312.347,Z 732.361,A -85,B 0,C 180,E1 -15703.15,E2 -15703.15} C_VEL
LIN {X 0,Y 311.791,Z 735.603,A -85,B 0,C 180,E1 -15704.969,E2 -15704.969} C_VEL
LIN {X 0,Y 311.19,Z 738.56,A -85,B 0,C 180,E1 -15707.35,E2 -15707.35} C_VEL
LIN {X 0,Y 310.912,Z 739.773,A -85,B 0,C 180,E1 -15709.041,E2 -15709.041} C_VEL
LIN {X 0,Y 310.743,Z 740.311,A -85,B 0,C 180,E1 -15710.709,E2 -15710.709} C_VEL
LIN {X 0,Y 310.676,Z 740.213,A -85,B 0,C 180,E1 -15712.355,E2 -15712.355} C_VEL
LIN {X 0,Y 310.772,Z 739.093,A -85,B 0,C 180,E1 -15714.5,E2 -15714.5} C_VEL
LIN {X 0,Y 311.057,Z 736.741,A -85,B 0,C 180,E1 -15716.716,E2 -15716.716} C_VEL
LIN {X 0,Y 311.55,Z 732.976,A -85,B 0,C 180,E1 -15719.003,E2 -15719.003} C_VEL
LIN {X 0,Y 312.222,Z 727.5,A -85,B 0,C 180,E1 -15721.386,E2 -15721.386} C_VEL
LIN {X 0,Y 313.005,Z 721.647,A -85,B 0,C 180,E1 -15723.317,E2 -15723.317} C_VEL
LIN {X 0,Y 313.948,Z 714.582,A -85,B 0,C 180,E1 -15725.183,E2 -15725.183} C_VEL
LIN {X 0,Y 315.115,Z 705.916,A -85,B 0,C 180,E1 -15727.027,E2 -15727.027} C_VEL
LIN {X 0,Y 316.342,Z 696.41,A -85,B 0,C 180,E1 -15728.661,E2 -15728.661} C_VEL
LIN {X 0,Y 317.561,Z 685.886,A -85,B 0,C 180,E1 -15730.107,E2 -15730.107} C_VEL
LIN {X 0,Y 318.822,Z 673.857,A -85,B 0,C 180,E1 -15731.417,E2 -15731.417} C_VEL
LIN {X 0,Y 319.806,Z 661.962,A -85,B 0,C 180,E1 -15732.413,E2 -15732.413} C_VEL
LIN {X 0,Y 320.599,Z 648.518,A -85,B 0,C 180,E1 -15733.238,E2 -15733.238} C_VEL
LIN {X 0,Y 321.169,Z 635.933,A -85,B 0,C 180,E1 -15733.754,E2 -15733.754} C_VEL
LIN {X 0,Y 323.232,Z 559.465,A -85,B 0,C 180,E1 -15735.568,E2 -15735.568} C_VEL
LIN {X 0,Y 317.554,Z 543.101,A -85,B 0,C 180,E1 -15736.38,E2 -15736.38} C_VEL
LIN {X 0,Y 313.461,Z 533.05,A -85,B 0,C 180,E1 -15736.941,E2 -15736.941} C_VEL
LIN {X 0,Y 312.657,Z 530.541,A -85,B 0,C 180,E1 -15737.093,E2 -15737.093} C_VEL
LIN {X 0,Y 312.829,Z 530.518,A -85,B 0,C 180,E1 -15741.298,E2 -15741.298} C_VEL
LIN {X 0,Y 312.9,Z 530.507,A -85,B 0,C 180,E1 -15743.552,E2 -15743.552} C_VEL
LIN {X 0,Y 312.935,Z 530.503,A -85,B 0,C 180,E1 -15747.426,E2 -15747.426} C_VEL
LIN {X 0,Y 313.1,Z 530.481,A -85,B 0,C 180,E1 -15750,E2 -15750} C_VEL
LIN {X 0,Y 312.935,Z 530.504,A -85,B 0,C 180,E1 -15752.574,E2 -15752.574} C_VEL
LIN {X 0,Y 312.907,Z 530.506,A -85,B 0,C 180,E1 -15756.448,E2 -15756.448} C_VEL
LIN {X 0,Y 312.785,Z 530.525,A -85,B 0,C 180,E1 -15759.049,E2 -15759.049} C_VEL
LIN {X 0,Y 312.632,Z 530.544,A -85,B 0,C 180,E1 -15762.991,E2 -15762.991} C_VEL
LIN {X 0,Y 312.635,Z 530.539,A -85,B 0,C 180,E1 -15765.65,E2 -15765.65} C_VEL
LIN {X 0,Y 312.627,Z 530.542,A -85,B 0,C 180,E1 -15769.236,E2 -15769.236} C_VEL
LIN {X 0,Y 312.542,Z 530.554,A -85,B 0,C 180,E1 -15772.789,E2 -15772.789} C_VEL
LIN {X 0,Y 312.598,Z 530.543,A -85,B 0,C 180,E1 -15775.935,E2 -15775.935} C_VEL
LIN {X 0,Y 312.542,Z 530.551,A -85,B 0,C 180,E1 -15779.649,E2 -15779.649} C_VEL
LIN {X 0,Y 312.515,Z 530.554,A -85,B 0,C 180,E1 -15783.689,E2 -15783.689} C_VEL
LIN {X 0,Y 312.548,Z 530.551,A -85,B 0,C 180,E1 -15787.381,E2 -15787.381} C_VEL
LIN {X 0,Y 312.529,Z 530.553,A -85,B 0,C 180,E1 -15790.702,E2 -15790.702} C_VEL
LIN {X 0,Y 312.589,Z 530.544,A -85,B 0,C 180,E1 -15794.184,E2 -15794.184} C_VEL
LIN {X 0,Y 312.544,Z 530.547,A -85,B 0,C 180,E1 -15797.364,E2 -15797.364} C_VEL
LIN {X 0,Y 311.896,Z 530.632,A -85,B 0,C 180,E1 -15798.439,E2 -15798.439} C_VEL
LIN {X 0,Y 309.007,Z 530.99,A -85,B 0,C 180,E1 -15800.187,E2 -15800.187} C_VEL
LIN {X 0,Y 306.563,Z 531.296,A -85,B 0,C 180,E1 -15801.605,E2 -15801.605} C_VEL
LIN {X 0,Y 305.544,Z 531.424,A -85,B 0,C 180,E1 -15802.704,E2 -15802.704} C_VEL
LIN {X 0,Y 305.479,Z 531.432,A -85,B 0,C 180,E1 -15803.076,E2 -15803.076} C_VEL
LIN {X 0,Y 305.458,Z 531.432,A -85,B 0,C 180,E1 -15806.483,E2 -15806.483} C_VEL
LIN {X 0,Y 305.489,Z 531.431,A -85,B 0,C 180,E1 -15810.95,E2 -15810.95} C_VEL
LIN {X 0,Y 305.564,Z 531.419,A -85,B 0,C 180,E1 -15814.088,E2 -15814.088} C_VEL
LIN {X 0,Y 305.473,Z 531.429,A -85,B 0,C 180,E1 -15818.402,E2 -15818.402} C_VEL
LIN {X 0,Y 305.572,Z 531.422,A -85,B 0,C 180,E1 -15821.217,E2 -15821.217} C_VEL
LIN {X 0,Y 305.641,Z 531.413,A -85,B 0,C 180,E1 -15825.349,E2 -15825.349} C_VEL
LIN {X 0,Y 305.633,Z 531.41,A -85,B 0,C 180,E1 -15829.4,E2 -15829.4} C_VEL
LIN {X 0,Y 305.806,Z 531.387,A -85,B 0,C 180,E1 -15832.075,E2 -15832.075} C_VEL
LIN {X 0,Y 305.686,Z 531.405,A -85,B 0,C 180,E1 -15834.724,E2 -15834.724} C_VEL
LIN {X 0,Y 305.952,Z 531.371,A -85,B 0,C 180,E1 -15838.684,E2 -15838.684} C_VEL
LIN {X 0,Y 305.956,Z 531.374,A -85,B 0,C 180,E1 -15841.317,E2 -15841.317} C_VEL
LIN {X 0,Y 305.687,Z 531.409,A -85,B 0,C 180,E1 -15845.277,E2 -15845.277} C_VEL
LIN {X 0,Y 305.791,Z 531.39,A -85,B 0,C 180,E1 -15847.927,E2 -15847.927} C_VEL
LIN {X 0,Y 305.597,Z 531.416,A -85,B 0,C 180,E1 -15851.946,E2 -15851.946} C_VEL
LIN {X 0,Y 305.632,Z 531.414,A -85,B 0,C 180,E1 -15855.036,E2 -15855.036} C_VEL
LIN {X 0,Y 305.572,Z 531.423,A -85,B 0,C 180,E1 -15859.446,E2 -15859.446} C_VEL
LIN {X 0,Y 305.486,Z 531.432,A -85,B 0,C 180,E1 -15863.042,E2 -15863.042} C_VEL
LIN {X 0,Y 305.543,Z 531.422,A -85,B 0,C 180,E1 -15866.228,E2 -15866.228} C_VEL
LIN {X 0,Y 305.493,Z 531.432,A -85,B 0,C 180,E1 -15869.051,E2 -15869.051} C_VEL
LIN {X 0,Y 305.444,Z 531.435,A -85,B 0,C 180,E1 -15871.953,E2 -15871.953} C_VEL
LIN {X 0,Y 305.46,Z 531.436,A -85,B 0,C 180,E1 -15875.114,E2 -15875.114} C_VEL
LIN {X 0,Y 305.447,Z 531.435,A -85,B 0,C 180,E1 -15878.53,E2 -15878.53} C_VEL
LIN {X 0,Y 305.461,Z 531.433,A -85,B 0,C 180,E1 -15882.589,E2 -15882.589} C_VEL
LIN {X 0,Y 305.489,Z 531.429,A -85,B 0,C 180,E1 -15886.358,E2 -15886.358} C_VEL
LIN {X 0,Y 305.484,Z 531.432,A -85,B 0,C 180,E1 -15889.898,E2 -15889.898} C_VEL
LIN {X 0,Y 305.502,Z 531.43,A -85,B 0,C 180,E1 -15893.627,E2 -15893.627} C_VEL
LIN {X 0,Y 305.533,Z 531.633,A -85,B 0,C 180,E1 -15895.823,E2 -15895.823} C_VEL
LIN {X 0,Y 308.231,Z 544.029,A -85,B 0,C 180,E1 -15899.515,E2 -15899.515} C_VEL
LIN {X 0,Y 310.428,Z 554.955,A -85,B 0,C 180,E1 -15902.613,E2 -15902.613} C_VEL
LIN {X 0,Y 309.713,Z 562.143,A -85,B 0,C 180,E1 -15904.46,E2 -15904.46} C_VEL
LIN {X 0,Y 309.577,Z 562.991,A -85,B 0,C 180,E1 -15904.674,E2 -15904.674} C_VEL
LIN {X 0,Y 315.573,Z 607.052,A -85,B 0,C 180,E1 -15906.263,E2 -15906.263} C_VEL
LIN {X 0,Y 314.017,Z 672.777,A -85,B 0,C 180,E1 -15907.897,E2 -15907.897} C_VEL
LIN {X 0,Y 313.152,Z 686.174,A -85,B 0,C 180,E1 -15908.482,E2 -15908.482} C_VEL
LIN {X 0,Y 311.966,Z 698.936,A -85,B 0,C 180,E1 -15909.305,E2 -15909.305} C_VEL
LIN {X 0,Y 310.726,Z 710.687,A -85,B 0,C 180,E1 -15910.34,E2 -15910.34} C_VEL
LIN {X 0,Y 309.255,Z 722.049,A -85,B 0,C 180,E1 -15911.62,E2 -15911.62} C_VEL
LIN {X 0,Y 307.984,Z 732.329,A -85,B 0,C 180,E1 -15913.086,E2 -15913.086} C_VEL
LIN {X 0,Y 306.846,Z 741.581,A -85,B 0,C 180,E1 -15914.729,E2 -15914.729} C_VEL
LIN {X 0,Y 305.64,Z 750.584,A -85,B 0,C 180,E1 -15916.707,E2 -15916.707} C_VEL
LIN {X 0,Y 304.669,Z 757.791,A -85,B 0,C 180,E1 -15918.693,E2 -15918.693} C_VEL
LIN {X 0,Y 304.174,Z 763.534,A -85,B 0,C 180,E1 -15920.693,E2 -15920.693} C_VEL
LIN {X 0,Y 303.853,Z 768.031,A -85,B 0,C 180,E1 -15922.692,E2 -15922.692} C_VEL
LIN {X 0,Y 303.747,Z 771.413,A -85,B 0,C 180,E1 -15924.69,E2 -15924.69} C_VEL
LIN {X 0,Y 303.779,Z 773.082,A -85,B 0,C 180,E1 -15926.02,E2 -15926.02} C_VEL
